KUKA KRL program: EPS_2_25252_SD4_A_20250910061725.src

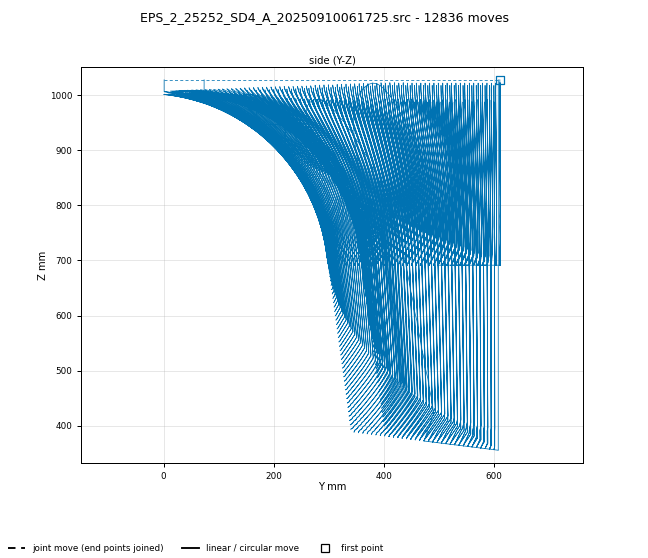
[picture p0: tool path of EPS_2_25252_SD4_A_20250910061725.src, 12836 of 12838 moves have a stored position in this frame; points joined in program order, loops and branches not executed]
&ACCESS RVP
&REL 4
&COMMENT QRS 19112012
&PARAM EDITMASK = *
DEF PART()
EXT BAS (BAS_COMMAND :IN,REAL :IN )
INT I
BAS (#INITMOV,0 )

;KUKA QRS Post kuka4.cps  Date:22-06-2017 !

File_ID=2825

QRS_PRE_INIT()

;Init var - Until changes are made in qrs_pre_init
Outlet_Square_prg=0
Inlet_1_Square_prg=0
Inlet_2_Square_prg=0
Inlet_3_Square_prg=0
Inlet_4_Square_prg=0
Inlet_5_Square_prg=0

Outlet_1={X 0.000, Y 400.000, Z 713.000, B 0.000, E1 0.000 }
Inlet_1={X 0.000, Y 400.000, Z 683.000, B 0.000, E1 208.000 }
Outlet_1_type=610
Inlet_1_type=610
;QRS#1=Sidecore dimensions
;QRS#2=600-24" Concrete
;QRS#3=600-24" Concrete
;QRS#4=
;QRS#5=
;QRS#6=
;QRS#7=
;QRS#8=
;QRS#9=S306-34L
;QRS#10=S306-34L
;QRS#11=
;QRS#12=
;QRS#13=
;QRS#14=
;QRS#15=
;QRS#16=1220x127x1372 4,5'
;QRS#17=EPS Height
;QRS#18=1018
;QRS#19=*
;QRS#20= UPDATED VERSION 22-06-2017
;QRS#21=*
Outlet_Square=0450
Inlet_1_Square=0450
Inlet_2_Square=0
Inlet_3_Square=0
Inlet_4_Square=0
Inlet_5_Square=0
Mill_Square=1
Outlet_Square_Prg=264
Inlet_1_Square_prg=264

QRS_INIT()

$ADVANCE=5

; T1
PTP {E1 178.274,E2 178.274}
PTP {X 0,Y 610.745,A -85,B 0,C 180,E1 178.274,E2 178.274,E3 0,E4 0,E5 0,E6 0}
QRS_SPEED_INIT()
LIN {X 0,Y 610.745,Z 1028,A -85,B 0,C 180,E1 178.274,E2 178.274,E3 0,E4 0,E5 0,E6 0} C_VEL
LIN {X 0,Y 610.745,Z 693.44,A -85,B 0,C 180,E1 178.274,E2 178.274} C_VEL
LIN {X 0,Y 610.771,Z 691.44,A -85,B 0,C 180,E1 178.462,E2 178.462} C_VEL
LIN {X 0,Y 611.874,Z 691.44,A -85,B 0,C 180,E1 181.167,E2 181.167} C_VEL
LIN {X 0,Y 611.801,Z 691.44,A -85,B 0,C 180,E1 188.197,E2 188.197} C_VEL
LIN {X 0,Y 611.817,Z 691.44,A -85,B 0,C 180,E1 195.354,E2 195.354} C_VEL
LIN {X 0,Y 611.765,Z 691.44,A -85,B 0,C 180,E1 202.769,E2 202.769} C_VEL
LIN {X 0,Y 611.741,Z 691.44,A -85,B 0,C 180,E1 210.614,E2 210.614} C_VEL
LIN {X 0,Y 610.574,Z 691.44,A -85,B 0,C 180,E1 217.262,E2 217.262} C_VEL
LIN {X 0,Y 611.71,Z 691.44,A -85,B 0,C 180,E1 219.162,E2 219.162} C_VEL
LIN {X 0,Y 610.308,Z 691.44,A -85,B 0,C 180,E1 222.361,E2 222.361} C_VEL
LIN {X 0,Y 610.623,Z 691.44,A -85,B 0,C 180,E1 225.583,E2 225.583} C_VEL
LIN {X 0,Y 611.712,Z 691.44,A -85,B 0,C 180,E1 227.765,E2 227.765} C_VEL
LIN {X 0,Y 611.694,Z 691.44,A -85,B 0,C 180,E1 235.934,E2 235.934} C_VEL
LIN {X 0,Y 611.734,Z 691.44,A -85,B 0,C 180,E1 236.288,E2 236.288} C_VEL
LIN {X 0,Y 610.695,Z 691.44,A -85,B 0,C 180,E1 236.459,E2 236.459} C_VEL
LIN {X 0,Y 610.433,Z 691.491,A -85,B 0,C 180,E1 236.481,E2 236.481} C_VEL
LIN {X 0,Y 611.42,Z 731.428,A -85,B 0,C 180,E1 237.097,E2 237.097} C_VEL
LIN {X 0,Y 611.517,Z 745.268,A -85,B 0,C 180,E1 237.335,E2 237.335} C_VEL
LIN {X 0,Y 611.325,Z 761.349,A -85,B 0,C 180,E1 237.681,E2 237.681} C_VEL
LIN {X 0,Y 611.672,Z 775.491,A -85,B 0,C 180,E1 238.087,E2 238.087} C_VEL
LIN {X 0,Y 611.736,Z 790.25,A -85,B 0,C 180,E1 238.571,E2 238.571} C_VEL
LIN {X 0,Y 611.693,Z 805.413,A -85,B 0,C 180,E1 239.145,E2 239.145} C_VEL
LIN {X 0,Y 611.448,Z 819.873,A -85,B 0,C 180,E1 239.763,E2 239.763} C_VEL
LIN {X 0,Y 611.625,Z 833.383,A -85,B 0,C 180,E1 240.435,E2 240.435} C_VEL
LIN {X 0,Y 611.599,Z 846.987,A -85,B 0,C 180,E1 241.179,E2 241.179} C_VEL
LIN {X 0,Y 611.634,Z 859.687,A -85,B 0,C 180,E1 241.947,E2 241.947} C_VEL
LIN {X 0,Y 611.641,Z 873.337,A -85,B 0,C 180,E1 242.859,E2 242.859} C_VEL
LIN {X 0,Y 611.572,Z 885.154,A -85,B 0,C 180,E1 243.716,E2 243.716} C_VEL
LIN {X 0,Y 611.333,Z 897.162,A -85,B 0,C 180,E1 244.66,E2 244.66} C_VEL
LIN {X 0,Y 611.276,Z 908.948,A -85,B 0,C 180,E1 245.678,E2 245.678} C_VEL
LIN {X 0,Y 611.472,Z 919.359,A -85,B 0,C 180,E1 246.662,E2 246.662} C_VEL
LIN {X 0,Y 611.734,Z 929.987,A -85,B 0,C 180,E1 247.753,E2 247.753} C_VEL
LIN {X 0,Y 611.445,Z 939.605,A -85,B 0,C 180,E1 248.799,E2 248.799} C_VEL
LIN {X 0,Y 611.088,Z 948.776,A -85,B 0,C 180,E1 249.876,E2 249.876} C_VEL
LIN {X 0,Y 611.074,Z 958.333,A -85,B 0,C 180,E1 251.115,E2 251.115} C_VEL
LIN {X 0,Y 611.399,Z 966.018,A -85,B 0,C 180,E1 252.202,E2 252.202} C_VEL
LIN {X 0,Y 611.821,Z 973.294,A -85,B 0,C 180,E1 253.324,E2 253.324} C_VEL
LIN {X 0,Y 611.107,Z 982.506,A -85,B 0,C 180,E1 254.862,E2 254.862} C_VEL
LIN {X 0,Y 610.739,Z 989.282,A -85,B 0,C 180,E1 256.13,E2 256.13} C_VEL
LIN {X 0,Y 610.875,Z 995.066,A -85,B 0,C 180,E1 257.336,E2 257.336} C_VEL
LIN {X 0,Y 611.566,Z 1001.375,A -85,B 0,C 180,E1 258.842,E2 258.842} C_VEL
LIN {X 0,Y 611.85,Z 1003.595,A -85,B 0,C 180,E1 259.441,E2 259.441} C_VEL
LIN {X 0,Y 611.525,Z 1005.814,A -85,B 0,C 180,E1 260.029,E2 260.029} C_VEL
LIN {X 0,Y 610.929,Z 1009.655,A -85,B 0,C 180,E1 261.204,E2 261.204} C_VEL
LIN {X 0,Y 610.672,Z 1012.99,A -85,B 0,C 180,E1 262.381,E2 262.381} C_VEL
LIN {X 0,Y 610.672,Z 1014.551,A -85,B 0,C 180,E1 262.97,E2 262.97} C_VEL
LIN {X 0,Y 611.06,Z 1017.123,A -85,B 0,C 180,E1 264.151,E2 264.151} C_VEL
LIN {X 0,Y 611.711,Z 1019.175,A -85,B 0,C 180,E1 265.329,E2 265.329} C_VEL
LIN {X 0,Y 611.37,Z 1020.807,A -85,B 0,C 180,E1 266.497,E2 266.497} C_VEL
LIN {X 0,Y 610.858,Z 1021.972,A -85,B 0,C 180,E1 267.634,E2 267.634} C_VEL
LIN {X 0,Y 610.688,Z 1022.778,A -85,B 0,C 180,E1 269.07,E2 269.07} C_VEL
LIN {X 0,Y 611.538,Z 1022.689,A -85,B 0,C 180,E1 271.17,E2 271.17} C_VEL
LIN {X 0,Y 611.319,Z 1021.671,A -85,B 0,C 180,E1 272.765,E2 272.765} C_VEL
LIN {X 0,Y 611.035,Z 1020.812,A -85,B 0,C 180,E1 273.51,E2 273.51} C_VEL
LIN {X 0,Y 610.805,Z 1019.194,A -85,B 0,C 180,E1 274.684,E2 274.684} C_VEL
LIN {X 0,Y 611.004,Z 1017.111,A -85,B 0,C 180,E1 275.855,E2 275.855} C_VEL
LIN {X 0,Y 611.55,Z 1014.527,A -85,B 0,C 180,E1 277.025,E2 277.025} C_VEL
LIN {X 0,Y 611.873,Z 1012.959,A -85,B 0,C 180,E1 277.61,E2 277.61} C_VEL
LIN {X 0,Y 611.24,Z 1009.637,A -85,B 0,C 180,E1 278.798,E2 278.798} C_VEL
LIN {X 0,Y 610.738,Z 1005.793,A -85,B 0,C 180,E1 279.99,E2 279.99} C_VEL
LIN {X 0,Y 610.738,Z 1000.147,A -85,B 0,C 180,E1 281.477,E2 281.477} C_VEL
LIN {X 0,Y 611.2,Z 995.039,A -85,B 0,C 180,E1 282.663,E2 282.663} C_VEL
LIN {X 0,Y 611.828,Z 989.347,A -85,B 0,C 180,E1 283.832,E2 283.832} C_VEL
LIN {X 0,Y 611.263,Z 982.264,A -85,B 0,C 180,E1 285.179,E2 285.179} C_VEL
LIN {X 0,Y 610.874,Z 973.74,A -85,B 0,C 180,E1 286.634,E2 286.634} C_VEL
LIN {X 0,Y 611.107,Z 964.915,A -85,B 0,C 180,E1 287.966,E2 287.966} C_VEL
LIN {X 0,Y 611.627,Z 956.003,A -85,B 0,C 180,E1 289.182,E2 289.182} C_VEL
LIN {X 0,Y 611.763,Z 951.154,A -85,B 0,C 180,E1 289.796,E2 289.796} C_VEL
LIN {X 0,Y 611.529,Z 944.981,A -85,B 0,C 180,E1 290.566,E2 290.566} C_VEL
LIN {X 0,Y 611.268,Z 937.362,A -85,B 0,C 180,E1 291.465,E2 291.465} C_VEL
LIN {X 0,Y 611.182,Z 926.922,A -85,B 0,C 180,E1 292.59,E2 292.59} C_VEL
LIN {X 0,Y 611.438,Z 916.306,A -85,B 0,C 180,E1 293.633,E2 293.633} C_VEL
LIN {X 0,Y 611.68,Z 905.113,A -85,B 0,C 180,E1 294.645,E2 294.645} C_VEL
LIN {X 0,Y 611.642,Z 894.625,A -85,B 0,C 180,E1 295.535,E2 295.535} C_VEL
LIN {X 0,Y 611.47,Z 882.903,A -85,B 0,C 180,E1 296.459,E2 296.459} C_VEL
LIN {X 0,Y 611.456,Z 869.526,A -85,B 0,C 180,E1 297.413,E2 297.413} C_VEL
LIN {X 0,Y 611.583,Z 857.642,A -85,B 0,C 180,E1 298.184,E2 298.184} C_VEL
LIN {X 0,Y 611.506,Z 843.831,A -85,B 0,C 180,E1 299.006,E2 299.006} C_VEL
LIN {X 0,Y 611.705,Z 829.665,A -85,B 0,C 180,E1 299.75,E2 299.75} C_VEL
LIN {X 0,Y 611.695,Z 816.017,A -85,B 0,C 180,E1 300.401,E2 300.401} C_VEL
LIN {X 0,Y 611.697,Z 800.985,A -85,B 0,C 180,E1 301.031,E2 301.031} C_VEL
LIN {X 0,Y 611.541,Z 786.836,A -85,B 0,C 180,E1 301.558,E2 301.558} C_VEL
LIN {X 0,Y 611.397,Z 780.445,A -85,B 0,C 180,E1 301.77,E2 301.77} C_VEL
LIN {X 0,Y 611.688,Z 770.796,A -85,B 0,C 180,E1 302.045,E2 302.045} C_VEL
LIN {X 0,Y 611.796,Z 757.518,A -85,B 0,C 180,E1 302.385,E2 302.385} C_VEL
LIN {X 0,Y 611.771,Z 741.883,A -85,B 0,C 180,E1 302.711,E2 302.711} C_VEL
LIN {X 0,Y 611.529,Z 722.323,A -85,B 0,C 180,E1 303.027,E2 303.027} C_VEL
LIN {X 0,Y 610.568,Z 694.458,A -85,B 0,C 180,E1 303.469,E2 303.469} C_VEL
LIN {X 0,Y 610.459,Z 691.44,A -85,B 0,C 180,E1 303.523,E2 303.523} C_VEL
LIN {X 0,Y 610.921,Z 691.44,A -85,B 0,C 180,E1 303.566,E2 303.566} C_VEL
LIN {X 0,Y 611.586,Z 691.44,A -85,B 0,C 180,E1 303.671,E2 303.671} C_VEL
LIN {X 0,Y 611.829,Z 691.44,A -85,B 0,C 180,E1 303.949,E2 303.949} C_VEL
LIN {X 0,Y 611.808,Z 691.44,A -85,B 0,C 180,E1 309.156,E2 309.156} C_VEL
LIN {X 0,Y 610.369,Z 691.44,A -85,B 0,C 180,E1 312.357,E2 312.357} C_VEL
LIN {X 0,Y 610.678,Z 691.44,A -85,B 0,C 180,E1 315.579,E2 315.579} C_VEL
LIN {X 0,Y 611.761,Z 691.44,A -85,B 0,C 180,E1 317.763,E2 317.763} C_VEL
LIN {X 0,Y 610.246,Z 691.44,A -85,B 0,C 180,E1 323.688,E2 323.688} C_VEL
LIN {X 0,Y 611.757,Z 691.44,A -85,B 0,C 180,E1 326.634,E2 326.634} C_VEL
LIN {X 0,Y 611.785,Z 691.44,A -85,B 0,C 180,E1 334.675,E2 334.675} C_VEL
LIN {X 0,Y 611.513,Z 691.44,A -85,B 0,C 180,E1 343.29,E2 343.29} C_VEL
LIN {X 0,Y 611.276,Z 691.44,A -85,B 0,C 180,E1 344.632,E2 344.632} C_VEL
LIN {X 0,Y 611.855,Z 691.44,A -85,B 0,C 180,E1 351.804,E2 351.804} C_VEL
LIN {X 0,Y 611.868,Z 691.44,A -85,B 0,C 180,E1 358.833,E2 358.833} C_VEL
LIN {X 0,Y 611.856,Z 691.44,A -85,B 0,C 180,E1 365.845,E2 365.845} C_VEL
LIN {X 0,Y 611.824,Z 691.44,A -85,B 0,C 180,E1 372.947,E2 372.947} C_VEL
LIN {X 0,Y 611.839,Z 691.44,A -85,B 0,C 180,E1 380.258,E2 380.258} C_VEL
LIN {X 0,Y 611.447,Z 691.44,A -85,B 0,C 180,E1 387.953,E2 387.953} C_VEL
LIN {X 0,Y 611.305,Z 691.44,A -85,B 0,C 180,E1 388.77,E2 388.77} C_VEL
LIN {X 0,Y 610.886,Z 691.44,A -85,B 0,C 180,E1 388.826,E2 388.826} C_VEL
LIN {X 0,Y 610.605,Z 692.257,A -85,B 0,C 180,E1 388.871,E2 388.871} C_VEL
LIN {X 0,Y 611.169,Z 709.751,A -85,B 0,C 180,E1 389.172,E2 389.172} C_VEL
LIN {X 0,Y 611.314,Z 717.452,A -85,B 0,C 180,E1 389.324,E2 389.324} C_VEL
LIN {X 0,Y 611.678,Z 731.173,A -85,B 0,C 180,E1 389.652,E2 389.652} C_VEL
LIN {X 0,Y 611.747,Z 746.429,A -85,B 0,C 180,E1 390.076,E2 390.076} C_VEL
LIN {X 0,Y 611.722,Z 761.243,A -85,B 0,C 180,E1 390.562,E2 390.562} C_VEL
LIN {X 0,Y 611.499,Z 775.09,A -85,B 0,C 180,E1 391.075,E2 391.075} C_VEL
LIN {X 0,Y 611.473,Z 779.918,A -85,B 0,C 180,E1 391.281,E2 391.281} C_VEL
LIN {X 0,Y 611.645,Z 790.127,A -85,B 0,C 180,E1 391.74,E2 391.74} C_VEL
LIN {X 0,Y 611.609,Z 803.759,A -85,B 0,C 180,E1 392.409,E2 392.409} C_VEL
LIN {X 0,Y 611.603,Z 816.719,A -85,B 0,C 180,E1 393.117,E2 393.117} C_VEL
LIN {X 0,Y 611.675,Z 830.91,A -85,B 0,C 180,E1 393.985,E2 393.985} C_VEL
LIN {X 0,Y 611.602,Z 842.971,A -85,B 0,C 180,E1 394.785,E2 394.785} C_VEL
LIN {X 0,Y 611.498,Z 854.83,A -85,B 0,C 180,E1 395.642,E2 395.642} C_VEL
LIN {X 0,Y 611.307,Z 867.776,A -85,B 0,C 180,E1 396.666,E2 396.666} C_VEL
LIN {X 0,Y 611.372,Z 878.558,A -85,B 0,C 180,E1 397.601,E2 397.601} C_VEL
LIN {X 0,Y 611.624,Z 890.243,A -85,B 0,C 180,E1 398.712,E2 398.712} C_VEL
LIN {X 0,Y 611.707,Z 898.191,A -85,B 0,C 180,E1 399.512,E2 399.512} C_VEL
LIN {X 0,Y 611.316,Z 909.19,A -85,B 0,C 180,E1 400.7,E2 400.7} C_VEL
LIN {X 0,Y 611.099,Z 918.7,A -85,B 0,C 180,E1 401.821,E2 401.821} C_VEL
LIN {X 0,Y 611.248,Z 927.831,A -85,B 0,C 180,E1 403.005,E2 403.005} C_VEL
LIN {X 0,Y 611.668,Z 936.135,A -85,B 0,C 180,E1 404.183,E2 404.183} C_VEL
LIN {X 0,Y 611.824,Z 939.64,A -85,B 0,C 180,E1 404.723,E2 404.723} C_VEL
LIN {X 0,Y 611.451,Z 944.743,A -85,B 0,C 180,E1 405.504,E2 405.504} C_VEL
LIN {X 0,Y 610.879,Z 952.592,A -85,B 0,C 180,E1 406.827,E2 406.827} C_VEL
LIN {X 0,Y 610.763,Z 958.932,A -85,B 0,C 180,E1 408.012,E2 408.012} C_VEL
LIN {X 0,Y 611.164,Z 965.191,A -85,B 0,C 180,E1 409.325,E2 409.325} C_VEL
LIN {X 0,Y 611.749,Z 970.163,A -85,B 0,C 180,E1 410.501,E2 410.501} C_VEL
LIN {X 0,Y 611.799,Z 971.533,A -85,B 0,C 180,E1 410.843,E2 410.843} C_VEL
LIN {X 0,Y 611.094,Z 976.54,A -85,B 0,C 180,E1 412.191,E2 412.191} C_VEL
LIN {X 0,Y 610.689,Z 981.321,A -85,B 0,C 180,E1 413.717,E2 413.717} C_VEL
LIN {X 0,Y 610.828,Z 984.007,A -85,B 0,C 180,E1 414.715,E2 414.715} C_VEL
LIN {X 0,Y 611.36,Z 986.671,A -85,B 0,C 180,E1 415.906,E2 415.906} C_VEL
LIN {X 0,Y 611.759,Z 988.072,A -85,B 0,C 180,E1 416.632,E2 416.632} C_VEL
LIN {X 0,Y 611.578,Z 989.364,A -85,B 0,C 180,E1 417.391,E2 417.391} C_VEL
LIN {X 0,Y 611.173,Z 990.338,A -85,B 0,C 180,E1 418.053,E2 418.053} C_VEL
LIN {X 0,Y 610.615,Z 991.788,A -85,B 0,C 180,E1 419.321,E2 419.321} C_VEL
LIN {X 0,Y 610.523,Z 992.469,A -85,B 0,C 180,E1 420.272,E2 420.272} C_VEL
LIN {X 0,Y 611.094,Z 992.97,A -85,B 0,C 180,E1 422.028,E2 422.028} C_VEL
LIN {X 0,Y 611.703,Z 992.701,A -85,B 0,C 180,E1 423.035,E2 423.035} C_VEL
LIN {X 0,Y 611.246,Z 991.725,A -85,B 0,C 180,E1 424.65,E2 424.65} C_VEL
LIN {X 0,Y 611.014,Z 990.672,A -85,B 0,C 180,E1 425.583,E2 425.583} C_VEL
LIN {X 0,Y 611.041,Z 989.261,A -85,B 0,C 180,E1 426.594,E2 426.594} C_VEL
LIN {X 0,Y 611.469,Z 986.875,A -85,B 0,C 180,E1 427.909,E2 427.909} C_VEL
LIN {X 0,Y 611.718,Z 985.672,A -85,B 0,C 180,E1 428.452,E2 428.452} C_VEL
LIN {X 0,Y 611.671,Z 984.243,A -85,B 0,C 180,E1 429.094,E2 429.094} C_VEL
LIN {X 0,Y 611.022,Z 980.931,A -85,B 0,C 180,E1 430.334,E2 430.334} C_VEL
LIN {X 0,Y 610.678,Z 976.08,A -85,B 0,C 180,E1 431.867,E2 431.867} C_VEL
LIN {X 0,Y 611.102,Z 970.181,A -85,B 0,C 180,E1 433.417,E2 433.417} C_VEL
LIN {X 0,Y 611.736,Z 964.877,A -85,B 0,C 180,E1 434.642,E2 434.642} C_VEL
LIN {X 0,Y 611.869,Z 963.707,A -85,B 0,C 180,E1 434.881,E2 434.881} C_VEL
LIN {X 0,Y 611.295,Z 957.857,A -85,B 0,C 180,E1 436.093,E2 436.093} C_VEL
LIN {X 0,Y 610.844,Z 951.248,A -85,B 0,C 180,E1 437.33,E2 437.33} C_VEL
LIN {X 0,Y 610.861,Z 944.132,A -85,B 0,C 180,E1 438.525,E2 438.525} C_VEL
LIN {X 0,Y 611.442,Z 934.12,A -85,B 0,C 180,E1 440.022,E2 440.022} C_VEL
LIN {X 0,Y 611.779,Z 927.636,A -85,B 0,C 180,E1 440.915,E2 440.915} C_VEL
LIN {X 0,Y 611.298,Z 916.221,A -85,B 0,C 180,E1 442.383,E2 442.383} C_VEL
LIN {X 0,Y 611.105,Z 907.499,A -85,B 0,C 180,E1 443.411,E2 443.411} C_VEL
LIN {X 0,Y 611.276,Z 896.469,A -85,B 0,C 180,E1 444.587,E2 444.587} C_VEL
LIN {X 0,Y 611.607,Z 885.785,A -85,B 0,C 180,E1 445.629,E2 445.629} C_VEL
LIN {X 0,Y 611.677,Z 874.98,A -85,B 0,C 180,E1 446.612,E2 446.612} C_VEL
LIN {X 0,Y 611.482,Z 863.577,A -85,B 0,C 180,E1 447.58,E2 447.58} C_VEL
LIN {X 0,Y 611.387,Z 852.606,A -85,B 0,C 180,E1 448.44,E2 448.44} C_VEL
LIN {X 0,Y 611.511,Z 840.572,A -85,B 0,C 180,E1 449.297,E2 449.297} C_VEL
LIN {X 0,Y 611.618,Z 828.032,A -85,B 0,C 180,E1 450.114,E2 450.114} C_VEL
LIN {X 0,Y 611.589,Z 820.26,A -85,B 0,C 180,E1 450.581,E2 450.581} C_VEL
LIN {X 0,Y 611.69,Z 812.057,A -85,B 0,C 180,E1 451.048,E2 451.048} C_VEL
LIN {X 0,Y 611.688,Z 799.787,A -85,B 0,C 180,E1 451.7,E2 451.7} C_VEL
LIN {X 0,Y 611.688,Z 786.561,A -85,B 0,C 180,E1 452.333,E2 452.333} C_VEL
LIN {X 0,Y 611.606,Z 770.8,A -85,B 0,C 180,E1 452.998,E2 452.998} C_VEL
LIN {X 0,Y 611.452,Z 760.468,A -85,B 0,C 180,E1 453.393,E2 453.393} C_VEL
LIN {X 0,Y 611.779,Z 742.741,A -85,B 0,C 180,E1 453.944,E2 453.944} C_VEL
LIN {X 0,Y 611.784,Z 726.733,A -85,B 0,C 180,E1 454.359,E2 454.359} C_VEL
LIN {X 0,Y 611.687,Z 711.157,A -85,B 0,C 180,E1 454.684,E2 454.684} C_VEL
LIN {X 0,Y 611.139,Z 694.076,A -85,B 0,C 180,E1 454.981,E2 454.981} C_VEL
LIN {X 0,Y 611.034,Z 691.44,A -85,B 0,C 180,E1 455.033,E2 455.033} C_VEL
LIN {X 0,Y 611.614,Z 691.44,A -85,B 0,C 180,E1 455.13,E2 455.13} C_VEL
LIN {X 0,Y 611.882,Z 691.44,A -85,B 0,C 180,E1 455.281,E2 455.281} C_VEL
LIN {X 0,Y 611.878,Z 691.44,A -85,B 0,C 180,E1 458.193,E2 458.193} C_VEL
LIN {X 0,Y 611.842,Z 691.44,A -85,B 0,C 180,E1 465.35,E2 465.35} C_VEL
LIN {X 0,Y 611.83,Z 691.44,A -85,B 0,C 180,E1 472.763,E2 472.763} C_VEL
LIN {X 0,Y 611.802,Z 691.44,A -85,B 0,C 180,E1 480.606,E2 480.606} C_VEL
LIN {X 0,Y 610.636,Z 691.44,A -85,B 0,C 180,E1 487.261,E2 487.261} C_VEL
LIN {X 0,Y 611.766,Z 691.44,A -85,B 0,C 180,E1 489.152,E2 489.152} C_VEL
LIN {X 0,Y 610.361,Z 691.44,A -85,B 0,C 180,E1 492.35,E2 492.35} C_VEL
LIN {X 0,Y 610.672,Z 691.44,A -85,B 0,C 180,E1 495.572,E2 495.572} C_VEL
LIN {X 0,Y 611.767,Z 691.44,A -85,B 0,C 180,E1 497.763,E2 497.763} C_VEL
LIN {X 0,Y 610.277,Z 691.44,A -85,B 0,C 180,E1 503.69,E2 503.69} C_VEL
LIN {X 0,Y 611.793,Z 691.44,A -85,B 0,C 180,E1 506.636,E2 506.636} C_VEL
LIN {X 0,Y 611.817,Z 691.44,A -85,B 0,C 180,E1 514.677,E2 514.677} C_VEL
LIN {X 0,Y 611.476,Z 691.44,A -85,B 0,C 180,E1 523.282,E2 523.282} C_VEL
LIN {X 0,Y 611.637,Z 691.44,A -85,B 0,C 180,E1 524.641,E2 524.641} C_VEL
LIN {X 0,Y 611.854,Z 691.44,A -85,B 0,C 180,E1 527.054,E2 527.054} C_VEL
LIN {X 0,Y 611.811,Z 691.44,A -85,B 0,C 180,E1 534.155,E2 534.155} C_VEL
LIN {X 0,Y 610.771,Z 691.44,A -85,B 0,C 180,E1 538.462,E2 538.462} C_VEL
LIN {X 0,Y 603.352,Z 691.44,A -85,B 0,C 180,E1 541.754,E2 541.754} C_VEL
LIN {X 0,Y 603.133,Z 691.44,A -85,B 0,C 180,E1 549.4,E2 549.4} C_VEL
LIN {X 0,Y 603.021,Z 691.44,A -85,B 0,C 180,E1 556.806,E2 556.806} C_VEL
LIN {X 0,Y 602.764,Z 691.44,A -85,B 0,C 180,E1 564.526,E2 564.526} C_VEL
LIN {X 0,Y 602.607,Z 691.44,A -85,B 0,C 180,E1 572.471,E2 572.471} C_VEL
LIN {X 0,Y 603.228,Z 691.44,A -85,B 0,C 180,E1 579.886,E2 579.886} C_VEL
LIN {X 0,Y 603.381,Z 691.44,A -85,B 0,C 180,E1 588.201,E2 588.201} C_VEL
LIN {X 0,Y 603.771,Z 692.599,A -85,B 0,C 180,E1 596.077,E2 596.077} C_VEL
LIN {X 0,Y 604.811,Z 776.815,A -85,B 0,C 180,E1 597.724,E2 597.724} C_VEL
LIN {X 0,Y 604.426,Z 842.241,A -85,B 0,C 180,E1 600.534,E2 600.534} C_VEL
LIN {X 0,Y 603.773,Z 901.578,A -85,B 0,C 180,E1 604.704,E2 604.704} C_VEL
LIN {X 0,Y 603.28,Z 950.003,A -85,B 0,C 180,E1 609.764,E2 609.764} C_VEL
LIN {X 0,Y 603.004,Z 985.712,A -85,B 0,C 180,E1 615.259,E2 615.259} C_VEL
LIN {X 0,Y 603.039,Z 1009.22,A -85,B 0,C 180,E1 620.95,E2 620.95} C_VEL
LIN {X 0,Y 603.404,Z 1020.765,A -85,B 0,C 180,E1 626.395,E2 626.395} C_VEL
LIN {X 0,Y 603.378,Z 1022.148,A -85,B 0,C 180,E1 632.162,E2 632.162} C_VEL
LIN {X 0,Y 603.3,Z 1010.379,A -85,B 0,C 180,E1 638.68,E2 638.68} C_VEL
LIN {X 0,Y 603.371,Z 983.789,A -85,B 0,C 180,E1 645.095,E2 645.095} C_VEL
LIN {X 0,Y 603.641,Z 943.759,A -85,B 0,C 180,E1 650.993,E2 650.993} C_VEL
LIN {X 0,Y 604.095,Z 892.092,A -85,B 0,C 180,E1 656.08,E2 656.08} C_VEL
LIN {X 0,Y 604.594,Z 831.211,A -85,B 0,C 180,E1 660.06,E2 660.06} C_VEL
LIN {X 0,Y 604.93,Z 766.154,A -85,B 0,C 180,E1 662.573,E2 662.573} C_VEL
LIN {X 0,Y 603.81,Z 691.44,A -85,B 0,C 180,E1 663.958,E2 663.958} C_VEL
LIN {X 0,Y 602.445,Z 691.44,A -85,B 0,C 180,E1 672.039,E2 672.039} C_VEL
LIN {X 0,Y 603.392,Z 691.44,A -85,B 0,C 180,E1 678.234,E2 678.234} C_VEL
LIN {X 0,Y 603.213,Z 691.44,A -85,B 0,C 180,E1 687.437,E2 687.437} C_VEL
LIN {X 0,Y 603.151,Z 691.44,A -85,B 0,C 180,E1 695.491,E2 695.491} C_VEL
LIN {X 0,Y 603.231,Z 691.44,A -85,B 0,C 180,E1 704.699,E2 704.699} C_VEL
LIN {X 0,Y 602.905,Z 691.44,A -85,B 0,C 180,E1 713.859,E2 713.859} C_VEL
LIN {X 0,Y 602.969,Z 691.44,A -85,B 0,C 180,E1 720.731,E2 720.731} C_VEL
LIN {X 0,Y 602.865,Z 691.44,A -85,B 0,C 180,E1 727.965,E2 727.965} C_VEL
LIN {X 0,Y 602.759,Z 691.44,A -85,B 0,C 180,E1 735.334,E2 735.334} C_VEL
LIN {X 0,Y 603.099,Z 691.44,A -85,B 0,C 180,E1 741.402,E2 741.402} C_VEL
LIN {X 0,Y 603.488,Z 692.92,A -85,B 0,C 180,E1 748.439,E2 748.439} C_VEL
LIN {X 0,Y 604.771,Z 763.762,A -85,B 0,C 180,E1 750.254,E2 750.254} C_VEL
LIN {X 0,Y 604.392,Z 826.547,A -85,B 0,C 180,E1 753.338,E2 753.338} C_VEL
LIN {X 0,Y 603.829,Z 884.4,A -85,B 0,C 180,E1 757.827,E2 757.827} C_VEL
LIN {X 0,Y 603.494,Z 931.716,A -85,B 0,C 180,E1 763.302,E2 763.302} C_VEL
LIN {X 0,Y 603.25,Z 966.27,A -85,B 0,C 180,E1 769.413,E2 769.413} C_VEL
LIN {X 0,Y 603.181,Z 986.033,A -85,B 0,C 180,E1 775.522,E2 775.522} C_VEL
LIN {X 0,Y 602.596,Z 992.687,A -85,B 0,C 180,E1 780.588,E2 780.588} C_VEL
LIN {X 0,Y 603.035,Z 990.881,A -85,B 0,C 180,E1 785.466,E2 785.466} C_VEL
LIN {X 0,Y 602.914,Z 980.226,A -85,B 0,C 180,E1 790.69,E2 790.69} C_VEL
LIN {X 0,Y 603.177,Z 956.506,A -85,B 0,C 180,E1 796.542,E2 796.542} C_VEL
LIN {X 0,Y 603.526,Z 918.219,A -85,B 0,C 180,E1 802.415,E2 802.415} C_VEL
LIN {X 0,Y 604.007,Z 865.701,A -85,B 0,C 180,E1 807.75,E2 807.75} C_VEL
LIN {X 0,Y 604.561,Z 805.25,A -85,B 0,C 180,E1 811.798,E2 811.798} C_VEL
LIN {X 0,Y 604.945,Z 742.287,A -85,B 0,C 180,E1 814.361,E2 814.361} C_VEL
LIN {X 0,Y 603.831,Z 691.44,A -85,B 0,C 180,E1 815.589,E2 815.589} C_VEL
LIN {X 0,Y 603.817,Z 691.44,A -85,B 0,C 180,E1 825.302,E2 825.302} C_VEL
LIN {X 0,Y 602.819,Z 691.44,A -85,B 0,C 180,E1 834.544,E2 834.544} C_VEL
LIN {X 0,Y 602.655,Z 691.44,A -85,B 0,C 180,E1 842.493,E2 842.493} C_VEL
LIN {X 0,Y 603.28,Z 691.44,A -85,B 0,C 180,E1 849.902,E2 849.902} C_VEL
LIN {X 0,Y 603.413,Z 691.44,A -85,B 0,C 180,E1 858.209,E2 858.209} C_VEL
LIN {X 0,Y 603.274,Z 691.44,A -85,B 0,C 180,E1 867.429,E2 867.429} C_VEL
LIN {X 0,Y 603.222,Z 691.44,A -85,B 0,C 180,E1 875.472,E2 875.472} C_VEL
LIN {X 0,Y 603.68,Z 691.44,A -85,B 0,C 180,E1 886.178,E2 886.178} C_VEL
LIN {X 0,Y 603.355,Z 691.44,A -85,B 0,C 180,E1 894.941,E2 894.941} C_VEL
LIN {X 0,Y 603.352,Z 691.44,A -85,B 0,C 180,E1 901.754,E2 901.754} C_VEL
LIN {X 0,Y 594.726,Z 691.44,A -85,B 0,C 180,E1 905.048,E2 905.048} C_VEL
LIN {X 0,Y 594.678,Z 691.44,A -85,B 0,C 180,E1 911.02,E2 911.02} C_VEL
LIN {X 0,Y 594.935,Z 691.44,A -85,B 0,C 180,E1 917.042,E2 917.042} C_VEL
LIN {X 0,Y 594.592,Z 691.44,A -85,B 0,C 180,E1 925.031,E2 925.031} C_VEL
LIN {X 0,Y 595.114,Z 691.44,A -85,B 0,C 180,E1 931.494,E2 931.494} C_VEL
LIN {X 0,Y 594.616,Z 691.44,A -85,B 0,C 180,E1 941.157,E2 941.157} C_VEL
LIN {X 0,Y 594.701,Z 691.44,A -85,B 0,C 180,E1 949.403,E2 949.403} C_VEL
LIN {X 0,Y 595.542,Z 692.888,A -85,B 0,C 180,E1 955.547,E2 955.547} C_VEL
LIN {X 0,Y 597.96,Z 779.246,A -85,B 0,C 180,E1 957.389,E2 957.389} C_VEL
LIN {X 0,Y 597.256,Z 843.942,A -85,B 0,C 180,E1 960.239,E2 960.239} C_VEL
LIN {X 0,Y 596.217,Z 903.96,A -85,B 0,C 180,E1 964.57,E2 964.57} C_VEL
LIN {X 0,Y 595.472,Z 951.481,A -85,B 0,C 180,E1 969.681,E2 969.681} C_VEL
LIN {X 0,Y 595.078,Z 986.267,A -85,B 0,C 180,E1 975.164,E2 975.164} C_VEL
LIN {X 0,Y 594.98,Z 1010.376,A -85,B 0,C 180,E1 981.197,E2 981.197} C_VEL
LIN {X 0,Y 595.416,Z 1020.765,A -85,B 0,C 180,E1 986.346,E2 986.346} C_VEL
LIN {X 0,Y 595.363,Z 1022.149,A -85,B 0,C 180,E1 992.191,E2 992.191} C_VEL
LIN {X 0,Y 595.255,Z 1010.378,A -85,B 0,C 180,E1 998.799,E2 998.799} C_VEL
LIN {X 0,Y 595.436,Z 984.428,A -85,B 0,C 180,E1 1005.178,E2 1005.178} C_VEL
LIN {X 0,Y 595.87,Z 945.376,A -85,B 0,C 180,E1 1011.084,E2 1011.084} C_VEL
LIN {X 0,Y 596.621,Z 893.819,A -85,B 0,C 180,E1 1016.292,E2 1016.292} C_VEL
LIN {X 0,Y 597.479,Z 832.394,A -85,B 0,C 180,E1 1020.391,E2 1020.391} C_VEL
LIN {X 0,Y 598.13,Z 767.802,A -85,B 0,C 180,E1 1022.944,E2 1022.944} C_VEL
LIN {X 0,Y 595.595,Z 691.44,A -85,B 0,C 180,E1 1024.496,E2 1024.496} C_VEL
LIN {X 0,Y 594.336,Z 691.44,A -85,B 0,C 180,E1 1032.582,E2 1032.582} C_VEL
LIN {X 0,Y 594.664,Z 691.44,A -85,B 0,C 180,E1 1039.431,E2 1039.431} C_VEL
LIN {X 0,Y 594.713,Z 691.44,A -85,B 0,C 180,E1 1048.483,E2 1048.483} C_VEL
LIN {X 0,Y 594.493,Z 691.44,A -85,B 0,C 180,E1 1056.712,E2 1056.712} C_VEL
LIN {X 0,Y 595.239,Z 691.44,A -85,B 0,C 180,E1 1064.488,E2 1064.488} C_VEL
LIN {X 0,Y 595.057,Z 691.44,A -85,B 0,C 180,E1 1073.422,E2 1073.422} C_VEL
LIN {X 0,Y 594.978,Z 691.44,A -85,B 0,C 180,E1 1080.74,E2 1080.74} C_VEL
LIN {X 0,Y 594.836,Z 691.44,A -85,B 0,C 180,E1 1088.074,E2 1088.074} C_VEL
LIN {X 0,Y 594.71,Z 691.44,A -85,B 0,C 180,E1 1095.546,E2 1095.546} C_VEL
LIN {X 0,Y 594.927,Z 691.44,A -85,B 0,C 180,E1 1101.711,E2 1101.711} C_VEL
LIN {X 0,Y 595.452,Z 692.462,A -85,B 0,C 180,E1 1107.919,E2 1107.919} C_VEL
LIN {X 0,Y 597.927,Z 761.951,A -85,B 0,C 180,E1 1109.778,E2 1109.778} C_VEL
LIN {X 0,Y 597.153,Z 825.254,A -85,B 0,C 180,E1 1112.878,E2 1112.878} C_VEL
LIN {X 0,Y 596.153,Z 881.742,A -85,B 0,C 180,E1 1117.242,E2 1117.242} C_VEL
LIN {X 0,Y 595.526,Z 928.799,A -85,B 0,C 180,E1 1122.623,E2 1122.623} C_VEL
LIN {X 0,Y 594.978,Z 962.977,A -85,B 0,C 180,E1 1128.498,E2 1128.498} C_VEL
LIN {X 0,Y 594.762,Z 982.401,A -85,B 0,C 180,E1 1133.904,E2 1133.904} C_VEL
LIN {X 0,Y 594.841,Z 991.25,A -85,B 0,C 180,E1 1138.709,E2 1138.709} C_VEL
LIN {X 0,Y 595.078,Z 991.348,A -85,B 0,C 180,E1 1145.116,E2 1145.116} C_VEL
LIN {X 0,Y 594.873,Z 979.906,A -85,B 0,C 180,E1 1150.912,E2 1150.912} C_VEL
LIN {X 0,Y 595.199,Z 956.552,A -85,B 0,C 180,E1 1156.734,E2 1156.734} C_VEL
LIN {X 0,Y 595.713,Z 918.317,A -85,B 0,C 180,E1 1162.682,E2 1162.682} C_VEL
LIN {X 0,Y 596.503,Z 865.85,A -85,B 0,C 180,E1 1168.087,E2 1168.087} C_VEL
LIN {X 0,Y 597.429,Z 805.396,A -85,B 0,C 180,E1 1172.184,E2 1172.184} C_VEL
LIN {X 0,Y 598.172,Z 742.236,A -85,B 0,C 180,E1 1174.776,E2 1174.776} C_VEL
LIN {X 0,Y 595.767,Z 691.646,A -85,B 0,C 180,E1 1175.982,E2 1175.982} C_VEL
LIN {X 0,Y 595.668,Z 691.44,A -85,B 0,C 180,E1 1185.516,E2 1185.516} C_VEL
LIN {X 0,Y 594.686,Z 691.44,A -85,B 0,C 180,E1 1194.902,E2 1194.902} C_VEL
LIN {X 0,Y 595.159,Z 691.44,A -85,B 0,C 180,E1 1201.516,E2 1201.516} C_VEL
LIN {X 0,Y 594.674,Z 691.44,A -85,B 0,C 180,E1 1211.172,E2 1211.172} C_VEL
LIN {X 0,Y 594.684,Z 691.44,A -85,B 0,C 180,E1 1219.407,E2 1219.407} C_VEL
LIN {X 0,Y 594.782,Z 691.44,A -85,B 0,C 180,E1 1228.463,E2 1228.463} C_VEL
LIN {X 0,Y 594.503,Z 691.44,A -85,B 0,C 180,E1 1236.69,E2 1236.69} C_VEL
LIN {X 0,Y 595.653,Z 691.44,A -85,B 0,C 180,E1 1245.988,E2 1245.988} C_VEL
LIN {X 0,Y 595.369,Z 691.44,A -85,B 0,C 180,E1 1254.873,E2 1254.873} C_VEL
LIN {X 0,Y 595.304,Z 691.44,A -85,B 0,C 180,E1 1262.181,E2 1262.181} C_VEL
LIN {X 0,Y 594.726,Z 691.44,A -85,B 0,C 180,E1 1265.048,E2 1265.048} C_VEL
LIN {X 0,Y 587.444,Z 691.44,A -85,B 0,C 180,E1 1268.415,E2 1268.415} C_VEL
LIN {X 0,Y 586.846,Z 691.44,A -85,B 0,C 180,E1 1277.284,E2 1277.284} C_VEL
LIN {X 0,Y 586.536,Z 691.44,A -85,B 0,C 180,E1 1285.251,E2 1285.251} C_VEL
LIN {X 0,Y 586.482,Z 691.44,A -85,B 0,C 180,E1 1292.756,E2 1292.756} C_VEL
LIN {X 0,Y 586.581,Z 691.44,A -85,B 0,C 180,E1 1301.248,E2 1301.248} C_VEL
LIN {X 0,Y 587.044,Z 691.44,A -85,B 0,C 180,E1 1308.76,E2 1308.76} C_VEL
LIN {X 0,Y 587.273,Z 693.317,A -85,B 0,C 180,E1 1314.998,E2 1314.998} C_VEL
LIN {X 0,Y 590.809,Z 705.891,A -85,B 0,C 180,E1 1315.42,E2 1315.42} C_VEL
LIN {X 0,Y 591.136,Z 781.262,A -85,B 0,C 180,E1 1317.032,E2 1317.032} C_VEL
LIN {X 0,Y 590.118,Z 844.997,A -85,B 0,C 180,E1 1319.902,E2 1319.902} C_VEL
LIN {X 0,Y 588.714,Z 903.961,A -85,B 0,C 180,E1 1324.222,E2 1324.222} C_VEL
LIN {X 0,Y 587.671,Z 952.959,A -85,B 0,C 180,E1 1329.597,E2 1329.597} C_VEL
LIN {X 0,Y 587.106,Z 987.674,A -85,B 0,C 180,E1 1335.231,E2 1335.231} C_VEL
LIN {X 0,Y 587.027,Z 1010.376,A -85,B 0,C 180,E1 1341.076,E2 1341.076} C_VEL
LIN {X 0,Y 587.425,Z 1020.766,A -85,B 0,C 180,E1 1346.297,E2 1346.297} C_VEL
LIN {X 0,Y 587.349,Z 1022.149,A -85,B 0,C 180,E1 1352.221,E2 1352.221} C_VEL
LIN {X 0,Y 587.22,Z 1010.378,A -85,B 0,C 180,E1 1358.92,E2 1358.92} C_VEL
LIN {X 0,Y 587.436,Z 984.431,A -85,B 0,C 180,E1 1365.39,E2 1365.39} C_VEL
LIN {X 0,Y 588.113,Z 946.08,A -85,B 0,C 180,E1 1371.289,E2 1371.289} C_VEL
LIN {X 0,Y 589.148,Z 894.983,A -85,B 0,C 180,E1 1376.556,E2 1376.556} C_VEL
LIN {X 0,Y 590.365,Z 833.851,A -85,B 0,C 180,E1 1380.715,E2 1380.715} C_VEL
LIN {X 0,Y 591.343,Z 769.887,A -85,B 0,C 180,E1 1383.313,E2 1383.313} C_VEL
LIN {X 0,Y 589.008,Z 696.086,A -85,B 0,C 180,E1 1384.844,E2 1384.844} C_VEL
LIN {X 0,Y 587.411,Z 691.44,A -85,B 0,C 180,E1 1385.154,E2 1385.154} C_VEL
LIN {X 0,Y 586.299,Z 691.44,A -85,B 0,C 180,E1 1393.309,E2 1393.309} C_VEL
LIN {X 0,Y 586.544,Z 691.44,A -85,B 0,C 180,E1 1399.752,E2 1399.752} C_VEL
LIN {X 0,Y 586.784,Z 691.44,A -85,B 0,C 180,E1 1408.007,E2 1408.007} C_VEL
LIN {X 0,Y 586.505,Z 691.44,A -85,B 0,C 180,E1 1416.717,E2 1416.717} C_VEL
LIN {X 0,Y 587.22,Z 691.44,A -85,B 0,C 180,E1 1424.271,E2 1424.271} C_VEL
LIN {X 0,Y 587.08,Z 691.44,A -85,B 0,C 180,E1 1433.333,E2 1433.333} C_VEL
LIN {X 0,Y 586.973,Z 691.44,A -85,B 0,C 180,E1 1440.751,E2 1440.751} C_VEL
LIN {X 0,Y 586.828,Z 691.44,A -85,B 0,C 180,E1 1448.184,E2 1448.184} C_VEL
LIN {X 0,Y 586.674,Z 691.44,A -85,B 0,C 180,E1 1455.765,E2 1455.765} C_VEL
LIN {X 0,Y 586.776,Z 691.44,A -85,B 0,C 180,E1 1462.028,E2 1462.028} C_VEL
LIN {X 0,Y 587.221,Z 692.727,A -85,B 0,C 180,E1 1467.378,E2 1467.378} C_VEL
LIN {X 0,Y 591.008,Z 708.683,A -85,B 0,C 180,E1 1467.885,E2 1467.885} C_VEL
LIN {X 0,Y 590.652,Z 776.585,A -85,B 0,C 180,E1 1469.924,E2 1469.924} C_VEL
LIN {X 0,Y 589.663,Z 840.532,A -85,B 0,C 180,E1 1473.508,E2 1473.508} C_VEL
LIN {X 0,Y 588.641,Z 895.645,A -85,B 0,C 180,E1 1478.314,E2 1478.314} C_VEL
LIN {X 0,Y 588.07,Z 940.626,A -85,B 0,C 180,E1 1484.158,E2 1484.158} C_VEL
LIN {X 0,Y 587.731,Z 971.385,A -85,B 0,C 180,E1 1490.34,E2 1490.34} C_VEL
LIN {X 0,Y 587.519,Z 989.187,A -85,B 0,C 180,E1 1497.073,E2 1497.073} C_VEL
LIN {X 0,Y 587.356,Z 992.744,A -85,B 0,C 180,E1 1503.118,E2 1503.118} C_VEL
LIN {X 0,Y 587.369,Z 983.756,A -85,B 0,C 180,E1 1509.586,E2 1509.586} C_VEL
LIN {X 0,Y 587.467,Z 960.261,A -85,B 0,C 180,E1 1516.176,E2 1516.176} C_VEL
LIN {X 0,Y 587.981,Z 922.578,A -85,B 0,C 180,E1 1522.399,E2 1522.399} C_VEL
LIN {X 0,Y 588.962,Z 873.251,A -85,B 0,C 180,E1 1527.785,E2 1527.785} C_VEL
LIN {X 0,Y 590.212,Z 813.78,A -85,B 0,C 180,E1 1532.119,E2 1532.119} C_VEL
LIN {X 0,Y 591.211,Z 749.734,A -85,B 0,C 180,E1 1534.97,E2 1534.97} C_VEL
LIN {X 0,Y 589.42,Z 696.366,A -85,B 0,C 180,E1 1536.332,E2 1536.332} C_VEL
LIN {X 0,Y 587.703,Z 691.44,A -85,B 0,C 180,E1 1536.673,E2 1536.673} C_VEL
LIN {X 0,Y 587.54,Z 691.44,A -85,B 0,C 180,E1 1545.737,E2 1545.737} C_VEL
LIN {X 0,Y 587.26,Z 691.44,A -85,B 0,C 180,E1 1553.613,E2 1553.613} C_VEL
LIN {X 0,Y 586.861,Z 691.44,A -85,B 0,C 180,E1 1562.014,E2 1562.014} C_VEL
LIN {X 0,Y 586.637,Z 691.44,A -85,B 0,C 180,E1 1571.275,E2 1571.275} C_VEL
LIN {X 0,Y 587.059,Z 691.44,A -85,B 0,C 180,E1 1578.766,E2 1578.766} C_VEL
LIN {X 0,Y 586.844,Z 691.44,A -85,B 0,C 180,E1 1587.986,E2 1587.986} C_VEL
LIN {X 0,Y 586.481,Z 691.44,A -85,B 0,C 180,E1 1596.724,E2 1596.724} C_VEL
LIN {X 0,Y 587.623,Z 691.44,A -85,B 0,C 180,E1 1605.792,E2 1605.792} C_VEL
LIN {X 0,Y 587.362,Z 691.44,A -85,B 0,C 180,E1 1614.803,E2 1614.803} C_VEL
LIN {X 0,Y 587.283,Z 691.44,A -85,B 0,C 180,E1 1622.211,E2 1622.211} C_VEL
LIN {X 0,Y 587.444,Z 691.44,A -85,B 0,C 180,E1 1628.415,E2 1628.415} C_VEL
LIN {X 0,Y 578.648,Z 691.44,A -85,B 0,C 180,E1 1631.801,E2 1631.801} C_VEL
LIN {X 0,Y 578.553,Z 691.44,A -85,B 0,C 180,E1 1639.123,E2 1639.123} C_VEL
LIN {X 0,Y 578.458,Z 691.44,A -85,B 0,C 180,E1 1645.629,E2 1645.629} C_VEL
LIN {X 0,Y 578.579,Z 691.44,A -85,B 0,C 180,E1 1652.502,E2 1652.502} C_VEL
LIN {X 0,Y 578.467,Z 691.44,A -85,B 0,C 180,E1 1661.609,E2 1661.609} C_VEL
LIN {X 0,Y 578.5,Z 691.44,A -85,B 0,C 180,E1 1670.005,E2 1670.005} C_VEL
LIN {X 0,Y 579.017,Z 693.387,A -85,B 0,C 180,E1 1674.425,E2 1674.425} C_VEL
LIN {X 0,Y 584.255,Z 707.854,A -85,B 0,C 180,E1 1675.004,E2 1675.004} C_VEL
LIN {X 0,Y 584.337,Z 783.354,A -85,B 0,C 180,E1 1676.67,E2 1676.67} C_VEL
LIN {X 0,Y 582.951,Z 846.472,A -85,B 0,C 180,E1 1679.586,E2 1679.586} C_VEL
LIN {X 0,Y 581.183,Z 906.713,A -85,B 0,C 180,E1 1684.113,E2 1684.113} C_VEL
LIN {X 0,Y 579.854,Z 954.534,A -85,B 0,C 180,E1 1689.522,E2 1689.522} C_VEL
LIN {X 0,Y 579.16,Z 988.548,A -85,B 0,C 180,E1 1695.198,E2 1695.198} C_VEL
LIN {X 0,Y 579.069,Z 1010.376,A -85,B 0,C 180,E1 1700.953,E2 1700.953} C_VEL
LIN {X 0,Y 579.433,Z 1020.766,A -85,B 0,C 180,E1 1706.245,E2 1706.245} C_VEL
LIN {X 0,Y 579.345,Z 1022.149,A -85,B 0,C 180,E1 1712.252,E2 1712.252} C_VEL
LIN {X 0,Y 579.188,Z 1010.378,A -85,B 0,C 180,E1 1719.045,E2 1719.045} C_VEL
LIN {X 0,Y 579.469,Z 984.614,A -85,B 0,C 180,E1 1725.571,E2 1725.571} C_VEL
LIN {X 0,Y 580.32,Z 946.182,A -85,B 0,C 180,E1 1731.576,E2 1731.576} C_VEL
LIN {X 0,Y 581.663,Z 894.352,A -85,B 0,C 180,E1 1736.978,E2 1736.978} C_VEL
LIN {X 0,Y 583.368,Z 833.326,A -85,B 0,C 180,E1 1741.154,E2 1741.154} C_VEL
LIN {X 0,Y 584.632,Z 769.889,A -85,B 0,C 180,E1 1743.747,E2 1743.747} C_VEL
LIN {X 0,Y 582.582,Z 699.439,A -85,B 0,C 180,E1 1745.235,E2 1745.235} C_VEL
LIN {X 0,Y 579.282,Z 691.44,A -85,B 0,C 180,E1 1745.702,E2 1745.702} C_VEL
LIN {X 0,Y 578.32,Z 691.44,A -85,B 0,C 180,E1 1754.058,E2 1754.058} C_VEL
LIN {X 0,Y 578.201,Z 691.44,A -85,B 0,C 180,E1 1760.739,E2 1760.739} C_VEL
LIN {X 0,Y 578.615,Z 691.44,A -85,B 0,C 180,E1 1768.474,E2 1768.474} C_VEL
LIN {X 0,Y 578.678,Z 691.44,A -85,B 0,C 180,E1 1776.036,E2 1776.036} C_VEL
LIN {X 0,Y 579.179,Z 691.44,A -85,B 0,C 180,E1 1784.047,E2 1784.047} C_VEL
LIN {X 0,Y 579.099,Z 691.44,A -85,B 0,C 180,E1 1793.24,E2 1793.24} C_VEL
LIN {X 0,Y 578.993,Z 691.44,A -85,B 0,C 180,E1 1800.761,E2 1800.761} C_VEL
LIN {X 0,Y 578.802,Z 691.44,A -85,B 0,C 180,E1 1808.299,E2 1808.299} C_VEL
LIN {X 0,Y 578.646,Z 691.44,A -85,B 0,C 180,E1 1815.989,E2 1815.989} C_VEL
LIN {X 0,Y 578.676,Z 691.44,A -85,B 0,C 180,E1 1822.353,E2 1822.353} C_VEL
LIN {X 0,Y 578.878,Z 692.199,A -85,B 0,C 180,E1 1826.799,E2 1826.799} C_VEL
LIN {X 0,Y 584.376,Z 709.046,A -85,B 0,C 180,E1 1827.45,E2 1827.45} C_VEL
LIN {X 0,Y 583.809,Z 776.552,A -85,B 0,C 180,E1 1829.502,E2 1829.502} C_VEL
LIN {X 0,Y 582.442,Z 839.667,A -85,B 0,C 180,E1 1833.061,E2 1833.061} C_VEL
LIN {X 0,Y 580.998,Z 895.557,A -85,B 0,C 180,E1 1837.974,E2 1837.974} C_VEL
LIN {X 0,Y 580.131,Z 940.469,A -85,B 0,C 180,E1 1843.88,E2 1843.88} C_VEL
LIN {X 0,Y 579.668,Z 971.12,A -85,B 0,C 180,E1 1850.103,E2 1850.103} C_VEL
LIN {X 0,Y 579.475,Z 988.47,A -85,B 0,C 180,E1 1856.557,E2 1856.557} C_VEL
LIN {X 0,Y 579.222,Z 992.841,A -85,B 0,C 180,E1 1862.709,E2 1862.709} C_VEL
LIN {X 0,Y 579.451,Z 984.708,A -85,B 0,C 180,E1 1869.295,E2 1869.295} C_VEL
LIN {X 0,Y 579.607,Z 962.03,A -85,B 0,C 180,E1 1875.984,E2 1875.984} C_VEL
LIN {X 0,Y 580.192,Z 925.457,A -85,B 0,C 180,E1 1882.296,E2 1882.296} C_VEL
LIN {X 0,Y 581.44,Z 875.46,A -85,B 0,C 180,E1 1887.944,E2 1887.944} C_VEL
LIN {X 0,Y 583.066,Z 817.005,A -85,B 0,C 180,E1 1892.331,E2 1892.331} C_VEL
LIN {X 0,Y 584.362,Z 752.85,A -85,B 0,C 180,E1 1895.302,E2 1895.302} C_VEL
LIN {X 0,Y 582.825,Z 699.51,A -85,B 0,C 180,E1 1896.729,E2 1896.729} C_VEL
LIN {X 0,Y 579.659,Z 691.44,A -85,B 0,C 180,E1 1897.144,E2 1897.144} C_VEL
LIN {X 0,Y 578.972,Z 691.44,A -85,B 0,C 180,E1 1906.948,E2 1906.948} C_VEL
LIN {X 0,Y 578.627,Z 691.44,A -85,B 0,C 180,E1 1915.217,E2 1915.217} C_VEL
LIN {X 0,Y 578.619,Z 691.44,A -85,B 0,C 180,E1 1922.526,E2 1922.526} C_VEL
LIN {X 0,Y 578.533,Z 691.44,A -85,B 0,C 180,E1 1931.624,E2 1931.624} C_VEL
LIN {X 0,Y 578.429,Z 691.44,A -85,B 0,C 180,E1 1940.004,E2 1940.004} C_VEL
LIN {X 0,Y 578.669,Z 691.44,A -85,B 0,C 180,E1 1948.467,E2 1948.467} C_VEL
LIN {X 0,Y 578.714,Z 691.44,A -85,B 0,C 180,E1 1956.015,E2 1956.015} C_VEL
LIN {X 0,Y 579.622,Z 691.44,A -85,B 0,C 180,E1 1965.592,E2 1965.592} C_VEL
LIN {X 0,Y 579.363,Z 691.44,A -85,B 0,C 180,E1 1974.731,E2 1974.731} C_VEL
LIN {X 0,Y 579.292,Z 691.44,A -85,B 0,C 180,E1 1982.241,E2 1982.241} C_VEL
LIN {X 0,Y 578.796,Z 691.44,A -85,B 0,C 180,E1 1990.502,E2 1990.502} C_VEL
LIN {X 0,Y 578.648,Z 691.44,A -85,B 0,C 180,E1 1991.801,E2 1991.801} C_VEL
LIN {X 0,Y 571.181,Z 691.44,A -85,B 0,C 180,E1 1995.275,E2 1995.275} C_VEL
LIN {X 0,Y 570.851,Z 691.44,A -85,B 0,C 180,E1 2004.314,E2 2004.314} C_VEL
LIN {X 0,Y 570.387,Z 691.44,A -85,B 0,C 180,E1 2013.059,E2 2013.059} C_VEL
LIN {X 0,Y 570.643,Z 691.44,A -85,B 0,C 180,E1 2020.717,E2 2020.717} C_VEL
LIN {X 0,Y 570.685,Z 691.44,A -85,B 0,C 180,E1 2029.344,E2 2029.344} C_VEL
LIN {X 0,Y 570.721,Z 693.215,A -85,B 0,C 180,E1 2033.824,E2 2033.824} C_VEL
LIN {X 0,Y 577.727,Z 709.32,A -85,B 0,C 180,E1 2034.572,E2 2034.572} C_VEL
LIN {X 0,Y 577.578,Z 783.433,A -85,B 0,C 180,E1 2036.23,E2 2036.23} C_VEL
LIN {X 0,Y 575.818,Z 847.483,A -85,B 0,C 180,E1 2039.233,E2 2039.233} C_VEL
LIN {X 0,Y 573.683,Z 906.341,A -85,B 0,C 180,E1 2043.714,E2 2043.714} C_VEL
LIN {X 0,Y 572.059,Z 955.568,A -85,B 0,C 180,E1 2049.374,E2 2049.374} C_VEL
LIN {X 0,Y 571.3,Z 988.547,A -85,B 0,C 180,E1 2054.989,E2 2054.989} C_VEL
LIN {X 0,Y 571.14,Z 1010.375,A -85,B 0,C 180,E1 2060.826,E2 2060.826} C_VEL
LIN {X 0,Y 571.44,Z 1020.766,A -85,B 0,C 180,E1 2066.193,E2 2066.193} C_VEL
LIN {X 0,Y 571.33,Z 1022.149,A -85,B 0,C 180,E1 2072.283,E2 2072.283} C_VEL
LIN {X 0,Y 571.474,Z 1012.354,A -85,B 0,C 180,E1 2078.398,E2 2078.398} C_VEL
LIN {X 0,Y 571.752,Z 988.549,A -85,B 0,C 180,E1 2084.998,E2 2084.998} C_VEL
LIN {X 0,Y 572.566,Z 949.052,A -85,B 0,C 180,E1 2091.506,E2 2091.506} C_VEL
LIN {X 0,Y 574.177,Z 898.145,A -85,B 0,C 180,E1 2097.018,E2 2097.018} C_VEL
LIN {X 0,Y 576.117,Z 839.493,A -85,B 0,C 180,E1 2101.231,E2 2101.231} C_VEL
LIN {X 0,Y 577.841,Z 774.251,A -85,B 0,C 180,E1 2104.069,E2 2104.069} C_VEL
LIN {X 0,Y 575.933,Z 701.814,A -85,B 0,C 180,E1 2105.668,E2 2105.668} C_VEL
LIN {X 0,Y 571.236,Z 691.44,A -85,B 0,C 180,E1 2106.29,E2 2106.29} C_VEL
LIN {X 0,Y 570.511,Z 691.44,A -85,B 0,C 180,E1 2115.212,E2 2115.212} C_VEL
LIN {X 0,Y 570.386,Z 691.44,A -85,B 0,C 180,E1 2124.242,E2 2124.242} C_VEL
LIN {X 0,Y 570.935,Z 691.44,A -85,B 0,C 180,E1 2134.008,E2 2134.008} C_VEL
LIN {X 0,Y 571.168,Z 691.44,A -85,B 0,C 180,E1 2143.817,E2 2143.817} C_VEL
LIN {X 0,Y 571.113,Z 691.44,A -85,B 0,C 180,E1 2153.145,E2 2153.145} C_VEL
LIN {X 0,Y 570.988,Z 691.44,A -85,B 0,C 180,E1 2160.772,E2 2160.772} C_VEL
LIN {X 0,Y 570.785,Z 691.44,A -85,B 0,C 180,E1 2168.416,E2 2168.416} C_VEL
LIN {X 0,Y 570.63,Z 691.44,A -85,B 0,C 180,E1 2176.22,E2 2176.22} C_VEL
LIN {X 0,Y 570.412,Z 691.44,A -85,B 0,C 180,E1 2183.383,E2 2183.383} C_VEL
LIN {X 0,Y 570.769,Z 692.928,A -85,B 0,C 180,E1 2186.235,E2 2186.235} C_VEL
LIN {X 0,Y 577.816,Z 711.639,A -85,B 0,C 180,E1 2187.047,E2 2187.047} C_VEL
LIN {X 0,Y 576.816,Z 779.338,A -85,B 0,C 180,E1 2189.187,E2 2189.187} C_VEL
LIN {X 0,Y 575.117,Z 842.478,A -85,B 0,C 180,E1 2192.864,E2 2192.864} C_VEL
LIN {X 0,Y 573.365,Z 898.025,A -85,B 0,C 180,E1 2197.902,E2 2197.902} C_VEL
LIN {X 0,Y 572.323,Z 942.993,A -85,B 0,C 180,E1 2204.04,E2 2204.04} C_VEL
LIN {X 0,Y 571.795,Z 973.712,A -85,B 0,C 180,E1 2210.678,E2 2210.678} C_VEL
LIN {X 0,Y 571.388,Z 989.314,A -85,B 0,C 180,E1 2217.012,E2 2217.012} C_VEL
LIN {X 0,Y 571.138,Z 992.318,A -85,B 0,C 180,E1 2223.997,E2 2223.997} C_VEL
LIN {X 0,Y 571.139,Z 982.772,A -85,B 0,C 180,E1 2230.198,E2 2230.198} C_VEL
LIN {X 0,Y 571.444,Z 960.13,A -85,B 0,C 180,E1 2236.613,E2 2236.613} C_VEL
LIN {X 0,Y 572.348,Z 922.784,A -85,B 0,C 180,E1 2242.956,E2 2242.956} C_VEL
LIN {X 0,Y 573.972,Z 873.542,A -85,B 0,C 180,E1 2248.485,E2 2248.485} C_VEL
LIN {X 0,Y 576,Z 814.049,A -85,B 0,C 180,E1 2252.926,E2 2252.926} C_VEL
LIN {X 0,Y 577.728,Z 749.78,A -85,B 0,C 180,E1 2255.843,E2 2255.843} C_VEL
LIN {X 0,Y 576.383,Z 702.368,A -85,B 0,C 180,E1 2257.126,E2 2257.126} C_VEL
LIN {X 0,Y 571.64,Z 691.44,A -85,B 0,C 180,E1 2257.771,E2 2257.771} C_VEL
LIN {X 0,Y 571.283,Z 691.44,A -85,B 0,C 180,E1 2266.197,E2 2266.197} C_VEL
LIN {X 0,Y 570.91,Z 691.44,A -85,B 0,C 180,E1 2274.332,E2 2274.332} C_VEL
LIN {X 0,Y 570.413,Z 691.44,A -85,B 0,C 180,E1 2283.077,E2 2283.077} C_VEL
LIN {X 0,Y 570.694,Z 691.44,A -85,B 0,C 180,E1 2290.731,E2 2290.731} C_VEL
LIN {X 0,Y 570.65,Z 691.44,A -85,B 0,C 180,E1 2299.345,E2 2299.345} C_VEL
LIN {X 0,Y 570.606,Z 691.44,A -85,B 0,C 180,E1 2308.76,E2 2308.76} C_VEL
LIN {X 0,Y 570.447,Z 691.44,A -85,B 0,C 180,E1 2316.611,E2 2316.611} C_VEL
LIN {X 0,Y 571.596,Z 691.44,A -85,B 0,C 180,E1 2325.715,E2 2325.715} C_VEL
LIN {X 0,Y 571.263,Z 691.44,A -85,B 0,C 180,E1 2335.012,E2 2335.012} C_VEL
LIN {X 0,Y 571.271,Z 691.44,A -85,B 0,C 180,E1 2342.273,E2 2342.273} C_VEL
LIN {X 0,Y 570.969,Z 691.44,A -85,B 0,C 180,E1 2349.934,E2 2349.934} C_VEL
LIN {X 0,Y 571.181,Z 691.44,A -85,B 0,C 180,E1 2355.275,E2 2355.275} C_VEL
LIN {X 0,Y 562.566,Z 691.44,A -85,B 0,C 180,E1 2358.76,E2 2358.76} C_VEL
LIN {X 0,Y 562.373,Z 691.44,A -85,B 0,C 180,E1 2366.418,E2 2366.418} C_VEL
LIN {X 0,Y 562.263,Z 691.44,A -85,B 0,C 180,E1 2373.568,E2 2373.568} C_VEL
LIN {X 0,Y 562.334,Z 691.44,A -85,B 0,C 180,E1 2382.084,E2 2382.084} C_VEL
LIN {X 0,Y 562.314,Z 691.44,A -85,B 0,C 180,E1 2390.637,E2 2390.637} C_VEL
LIN {X 0,Y 562.467,Z 692.61,A -85,B 0,C 180,E1 2393.198,E2 2393.198} C_VEL
LIN {X 0,Y 571.261,Z 712.961,A -85,B 0,C 180,E1 2394.164,E2 2394.164} C_VEL
LIN {X 0,Y 570.841,Z 785.484,A -85,B 0,C 180,E1 2395.849,E2 2395.849} C_VEL
LIN {X 0,Y 568.708,Z 848.629,A -85,B 0,C 180,E1 2398.881,E2 2398.881} C_VEL
LIN {X 0,Y 566.139,Z 908.341,A -85,B 0,C 180,E1 2403.535,E2 2403.535} C_VEL
LIN {X 0,Y 564.323,Z 955.9,A -85,B 0,C 180,E1 2409.125,E2 2409.125} C_VEL
LIN {X 0,Y 563.284,Z 990.328,A -85,B 0,C 180,E1 2415.17,E2 2415.17} C_VEL
LIN {X 0,Y 563.196,Z 1010.375,A -85,B 0,C 180,E1 2420.695,E2 2420.695} C_VEL
LIN {X 0,Y 563.471,Z 1020.766,A -85,B 0,C 180,E1 2426.139,E2 2426.139} C_VEL
LIN {X 0,Y 563.315,Z 1022.149,A -85,B 0,C 180,E1 2432.316,E2 2432.316} C_VEL
LIN {X 0,Y 563.418,Z 1012.355,A -85,B 0,C 180,E1 2438.519,E2 2438.519} C_VEL
LIN {X 0,Y 563.77,Z 988.548,A -85,B 0,C 180,E1 2445.216,E2 2445.216} C_VEL
LIN {X 0,Y 564.791,Z 950.028,A -85,B 0,C 180,E1 2451.68,E2 2451.68} C_VEL
LIN {X 0,Y 566.707,Z 899.297,A -85,B 0,C 180,E1 2457.296,E2 2457.296} C_VEL
LIN {X 0,Y 569.067,Z 840.634,A -85,B 0,C 180,E1 2461.595,E2 2461.595} C_VEL
LIN {X 0,Y 571.101,Z 775.946,A -85,B 0,C 180,E1 2464.468,E2 2464.468} C_VEL
LIN {X 0,Y 569.695,Z 705.561,A -85,B 0,C 180,E1 2466.062,E2 2466.062} C_VEL
LIN {X 0,Y 563.148,Z 691.44,A -85,B 0,C 180,E1 2466.947,E2 2466.947} C_VEL
LIN {X 0,Y 562.834,Z 691.44,A -85,B 0,C 180,E1 2477.858,E2 2477.858} C_VEL
LIN {X 0,Y 562.569,Z 691.44,A -85,B 0,C 180,E1 2488.287,E2 2488.287} C_VEL
LIN {X 0,Y 562.326,Z 691.44,A -85,B 0,C 180,E1 2496.983,E2 2496.983} C_VEL
LIN {X 0,Y 562.829,Z 691.44,A -85,B 0,C 180,E1 2505.174,E2 2505.174} C_VEL
LIN {X 0,Y 563.122,Z 691.44,A -85,B 0,C 180,E1 2513.048,E2 2513.048} C_VEL
LIN {X 0,Y 562.989,Z 691.44,A -85,B 0,C 180,E1 2520.783,E2 2520.783} C_VEL
LIN {X 0,Y 562.765,Z 691.44,A -85,B 0,C 180,E1 2528.537,E2 2528.537} C_VEL
LIN {X 0,Y 562.64,Z 691.44,A -85,B 0,C 180,E1 2536.759,E2 2536.759} C_VEL
LIN {X 0,Y 562.416,Z 691.44,A -85,B 0,C 180,E1 2545.319,E2 2545.319} C_VEL
LIN {X 0,Y 565.479,Z 698.691,A -85,B 0,C 180,E1 2545.938,E2 2545.938} C_VEL
LIN {X 0,Y 571.241,Z 714.152,A -85,B 0,C 180,E1 2546.637,E2 2546.637} C_VEL
LIN {X 0,Y 569.836,Z 782.848,A -85,B 0,C 180,E1 2548.9,E2 2548.9} C_VEL
LIN {X 0,Y 567.782,Z 845.054,A -85,B 0,C 180,E1 2552.655,E2 2552.655} C_VEL
LIN {X 0,Y 565.7,Z 899.678,A -85,B 0,C 180,E1 2557.75,E2 2557.75} C_VEL
LIN {X 0,Y 564.421,Z 943.699,A -85,B 0,C 180,E1 2563.904,E2 2563.904} C_VEL
LIN {X 0,Y 563.777,Z 974.554,A -85,B 0,C 180,E1 2570.76,E2 2570.76} C_VEL
LIN {X 0,Y 563.307,Z 989.884,A -85,B 0,C 180,E1 2577.324,E2 2577.324} C_VEL
LIN {X 0,Y 563.061,Z 991.991,A -85,B 0,C 180,E1 2584.525,E2 2584.525} C_VEL
LIN {X 0,Y 562.988,Z 981.705,A -85,B 0,C 180,E1 2590.75,E2 2590.75} C_VEL
LIN {X 0,Y 563.457,Z 960.397,A -85,B 0,C 180,E1 2596.766,E2 2596.766} C_VEL
LIN {X 0,Y 564.546,Z 924.275,A -85,B 0,C 180,E1 2603.052,E2 2603.052} C_VEL
LIN {X 0,Y 566.492,Z 874.715,A -85,B 0,C 180,E1 2608.753,E2 2608.753} C_VEL
LIN {X 0,Y 568.901,Z 815.734,A -85,B 0,C 180,E1 2613.25,E2 2613.25} C_VEL
LIN {X 0,Y 570.976,Z 751.957,A -85,B 0,C 180,E1 2616.222,E2 2616.222} C_VEL
LIN {X 0,Y 570.011,Z 705.626,A -85,B 0,C 180,E1 2617.522,E2 2617.522} C_VEL
LIN {X 0,Y 563.603,Z 691.44,A -85,B 0,C 180,E1 2618.271,E2 2618.271} C_VEL
LIN {X 0,Y 562.981,Z 691.44,A -85,B 0,C 180,E1 2626.904,E2 2626.904} C_VEL
LIN {X 0,Y 562.578,Z 691.44,A -85,B 0,C 180,E1 2635.372,E2 2635.372} C_VEL
LIN {X 0,Y 562.298,Z 691.44,A -85,B 0,C 180,E1 2643.592,E2 2643.592} C_VEL
LIN {X 0,Y 562.374,Z 691.44,A -85,B 0,C 180,E1 2652.096,E2 2652.096} C_VEL
LIN {X 0,Y 562.343,Z 691.44,A -85,B 0,C 180,E1 2660.276,E2 2660.276} C_VEL
LIN {X 0,Y 562.624,Z 691.44,A -85,B 0,C 180,E1 2668.266,E2 2668.266} C_VEL
LIN {X 0,Y 562.321,Z 691.44,A -85,B 0,C 180,E1 2676.96,E2 2676.96} C_VEL
LIN {X 0,Y 563.511,Z 691.44,A -85,B 0,C 180,E1 2686.761,E2 2686.761} C_VEL
LIN {X 0,Y 562.94,Z 691.44,A -85,B 0,C 180,E1 2696.126,E2 2696.126} C_VEL
LIN {X 0,Y 562.822,Z 691.44,A -85,B 0,C 180,E1 2703.853,E2 2703.853} C_VEL
LIN {X 0,Y 562.649,Z 691.44,A -85,B 0,C 180,E1 2711.656,E2 2711.656} C_VEL
LIN {X 0,Y 562.566,Z 691.44,A -85,B 0,C 180,E1 2718.76,E2 2718.76} C_VEL
LIN {X 0,Y 554.858,Z 691.44,A -85,B 0,C 180,E1 2722.306,E2 2722.306} C_VEL
LIN {X 0,Y 554.553,Z 691.44,A -85,B 0,C 180,E1 2732.226,E2 2732.226} C_VEL
LIN {X 0,Y 554.463,Z 691.44,A -85,B 0,C 180,E1 2741.176,E2 2741.176} C_VEL
LIN {X 0,Y 554.436,Z 691.44,A -85,B 0,C 180,E1 2749.966,E2 2749.966} C_VEL
LIN {X 0,Y 554.496,Z 693.381,A -85,B 0,C 180,E1 2752.591,E2 2752.591} C_VEL
LIN {X 0,Y 564.774,Z 714.733,A -85,B 0,C 180,E1 2753.715,E2 2753.715} C_VEL
LIN {X 0,Y 564.145,Z 786.079,A -85,B 0,C 180,E1 2755.408,E2 2755.408} C_VEL
LIN {X 0,Y 561.65,Z 849.487,A -85,B 0,C 180,E1 2758.503,E2 2758.503} C_VEL
LIN {X 0,Y 558.757,Z 908.408,A -85,B 0,C 180,E1 2763.164,E2 2763.164} C_VEL
LIN {X 0,Y 556.515,Z 957.348,A -85,B 0,C 180,E1 2769.028,E2 2769.028} C_VEL
LIN {X 0,Y 555.389,Z 990.33,A -85,B 0,C 180,E1 2774.954,E2 2774.954} C_VEL
LIN {X 0,Y 555.266,Z 1010.374,A -85,B 0,C 180,E1 2780.561,E2 2780.561} C_VEL
LIN {X 0,Y 555.477,Z 1020.766,A -85,B 0,C 180,E1 2786.083,E2 2786.083} C_VEL
LIN {X 0,Y 555.301,Z 1022.15,A -85,B 0,C 180,E1 2792.349,E2 2792.349} C_VEL
LIN {X 0,Y 555.365,Z 1012.355,A -85,B 0,C 180,E1 2798.644,E2 2798.644} C_VEL
LIN {X 0,Y 555.773,Z 988.547,A -85,B 0,C 180,E1 2805.44,E2 2805.44} C_VEL
LIN {X 0,Y 557.026,Z 950.549,A -85,B 0,C 180,E1 2811.924,E2 2811.924} C_VEL
LIN {X 0,Y 559.288,Z 899.883,A -85,B 0,C 180,E1 2817.633,E2 2817.633} C_VEL
LIN {X 0,Y 562.028,Z 841.889,A -85,B 0,C 180,E1 2821.962,E2 2821.962} C_VEL
LIN {X 0,Y 564.383,Z 777.522,A -85,B 0,C 180,E1 2824.881,E2 2824.881} C_VEL
LIN {X 0,Y 563.371,Z 708.807,A -85,B 0,C 180,E1 2826.482,E2 2826.482} C_VEL
LIN {X 0,Y 555.102,Z 691.44,A -85,B 0,C 180,E1 2827.542,E2 2827.542} C_VEL
LIN {X 0,Y 554.813,Z 691.44,A -85,B 0,C 180,E1 2837.954,E2 2837.954} C_VEL
LIN {X 0,Y 554.596,Z 691.44,A -85,B 0,C 180,E1 2847.777,E2 2847.777} C_VEL
LIN {X 0,Y 554.382,Z 691.44,A -85,B 0,C 180,E1 2856.634,E2 2856.634} C_VEL
LIN {X 0,Y 554.839,Z 691.44,A -85,B 0,C 180,E1 2864.956,E2 2864.956} C_VEL
LIN {X 0,Y 555.134,Z 691.44,A -85,B 0,C 180,E1 2872.947,E2 2872.947} C_VEL
LIN {X 0,Y 554.984,Z 691.44,A -85,B 0,C 180,E1 2880.794,E2 2880.794} C_VEL
LIN {X 0,Y 554.777,Z 691.44,A -85,B 0,C 180,E1 2888.661,E2 2888.661} C_VEL
LIN {X 0,Y 554.637,Z 691.44,A -85,B 0,C 180,E1 2896.701,E2 2896.701} C_VEL
LIN {X 0,Y 554.42,Z 692.37,A -85,B 0,C 180,E1 2905.002,E2 2905.002} C_VEL
LIN {X 0,Y 564.694,Z 716.266,A -85,B 0,C 180,E1 2906.213,E2 2906.213} C_VEL
LIN {X 0,Y 562.955,Z 785.328,A -85,B 0,C 180,E1 2908.561,E2 2908.561} C_VEL
LIN {X 0,Y 560.468,Z 847.254,A -85,B 0,C 180,E1 2912.412,E2 2912.412} C_VEL
LIN {X 0,Y 558.032,Z 901.189,A -85,B 0,C 180,E1 2917.576,E2 2917.576} C_VEL
LIN {X 0,Y 556.516,Z 944.203,A -85,B 0,C 180,E1 2923.727,E2 2923.727} C_VEL
LIN {X 0,Y 555.834,Z 974.69,A -85,B 0,C 180,E1 2930.637,E2 2930.637} C_VEL
LIN {X 0,Y 555.194,Z 990.514,A -85,B 0,C 180,E1 2937.791,E2 2937.791} C_VEL
LIN {X 0,Y 555.047,Z 991.756,A -85,B 0,C 180,E1 2944.926,E2 2944.926} C_VEL
LIN {X 0,Y 554.919,Z 981.091,A -85,B 0,C 180,E1 2951.125,E2 2951.125} C_VEL
LIN {X 0,Y 555.422,Z 958.684,A -85,B 0,C 180,E1 2957.374,E2 2957.374} C_VEL
LIN {X 0,Y 556.776,Z 922.772,A -85,B 0,C 180,E1 2963.575,E2 2963.575} C_VEL
LIN {X 0,Y 559.084,Z 873.823,A -85,B 0,C 180,E1 2969.223,E2 2969.223} C_VEL
LIN {X 0,Y 561.915,Z 815.82,A -85,B 0,C 180,E1 2973.678,E2 2973.678} C_VEL
LIN {X 0,Y 564.276,Z 752.698,A -85,B 0,C 180,E1 2976.661,E2 2976.661} C_VEL
LIN {X 0,Y 563.411,Z 708.477,A -85,B 0,C 180,E1 2977.951,E2 2977.951} C_VEL
LIN {X 0,Y 555.288,Z 691.44,A -85,B 0,C 180,E1 2979.042,E2 2979.042} C_VEL
LIN {X 0,Y 555.083,Z 691.44,A -85,B 0,C 180,E1 2986.683,E2 2986.683} C_VEL
LIN {X 0,Y 554.672,Z 691.44,A -85,B 0,C 180,E1 2995.093,E2 2995.093} C_VEL
LIN {X 0,Y 554.339,Z 691.44,A -85,B 0,C 180,E1 3003.397,E2 3003.397} C_VEL
LIN {X 0,Y 554.379,Z 691.44,A -85,B 0,C 180,E1 3012.12,E2 3012.12} C_VEL
LIN {X 0,Y 554.391,Z 691.44,A -85,B 0,C 180,E1 3019.966,E2 3019.966} C_VEL
LIN {X 0,Y 554.649,Z 691.44,A -85,B 0,C 180,E1 3027.755,E2 3027.755} C_VEL
LIN {X 0,Y 554.385,Z 691.44,A -85,B 0,C 180,E1 3036.611,E2 3036.611} C_VEL
LIN {X 0,Y 555.49,Z 691.44,A -85,B 0,C 180,E1 3046.566,E2 3046.566} C_VEL
LIN {X 0,Y 554.961,Z 691.44,A -85,B 0,C 180,E1 3056.071,E2 3056.071} C_VEL
LIN {X 0,Y 554.841,Z 691.44,A -85,B 0,C 180,E1 3063.909,E2 3063.909} C_VEL
LIN {X 0,Y 554.65,Z 691.44,A -85,B 0,C 180,E1 3071.827,E2 3071.827} C_VEL
LIN {X 0,Y 554.605,Z 691.44,A -85,B 0,C 180,E1 3079.983,E2 3079.983} C_VEL
LIN {X 0,Y 554.858,Z 691.44,A -85,B 0,C 180,E1 3082.306,E2 3082.306} C_VEL
LIN {X 0,Y 546.458,Z 691.44,A -85,B 0,C 180,E1 3085.891,E2 3085.891} C_VEL
LIN {X 0,Y 546.405,Z 691.44,A -85,B 0,C 180,E1 3092.766,E2 3092.766} C_VEL
LIN {X 0,Y 546.516,Z 691.44,A -85,B 0,C 180,E1 3100.703,E2 3100.703} C_VEL
LIN {X 0,Y 546.485,Z 691.44,A -85,B 0,C 180,E1 3109.748,E2 3109.748} C_VEL
LIN {X 0,Y 546.468,Z 693.431,A -85,B 0,C 180,E1 3111.945,E2 3111.945} C_VEL
LIN {X 0,Y 558.381,Z 718.426,A -85,B 0,C 180,E1 3113.29,E2 3113.29} C_VEL
LIN {X 0,Y 557.451,Z 788.05,A -85,B 0,C 180,E1 3115.004,E2 3115.004} C_VEL
LIN {X 0,Y 554.489,Z 852.327,A -85,B 0,C 180,E1 3118.241,E2 3118.241} C_VEL
LIN {X 0,Y 551.224,Z 910.444,A -85,B 0,C 180,E1 3122.982,E2 3122.982} C_VEL
LIN {X 0,Y 548.837,Z 957.348,A -85,B 0,C 180,E1 3128.72,E2 3128.72} C_VEL
LIN {X 0,Y 547.413,Z 991.402,A -85,B 0,C 180,E1 3134.98,E2 3134.98} C_VEL
LIN {X 0,Y 546.987,Z 1012.354,A -85,B 0,C 180,E1 3141.222,E2 3141.222} C_VEL
LIN {X 0,Y 546.921,Z 1022.149,A -85,B 0,C 180,E1 3147.614,E2 3147.614} C_VEL
LIN {X 0,Y 547.032,Z 1020.768,A -85,B 0,C 180,E1 3153.977,E2 3153.977} C_VEL
LIN {X 0,Y 546.926,Z 1008.898,A -85,B 0,C 180,E1 3160.101,E2 3160.101} C_VEL
LIN {X 0,Y 547.651,Z 984.619,A -85,B 0,C 180,E1 3166.501,E2 3166.501} C_VEL
LIN {X 0,Y 549.322,Z 947.327,A -85,B 0,C 180,E1 3172.707,E2 3172.707} C_VEL
LIN {X 0,Y 552.156,Z 895.461,A -85,B 0,C 180,E1 3178.448,E2 3178.448} C_VEL
LIN {X 0,Y 555.467,Z 835.315,A -85,B 0,C 180,E1 3182.788,E2 3182.788} C_VEL
LIN {X 0,Y 558.06,Z 771.915,A -85,B 0,C 180,E1 3185.528,E2 3185.528} C_VEL
LIN {X 0,Y 556.765,Z 711.26,A -85,B 0,C 180,E1 3186.947,E2 3186.947} C_VEL
LIN {X 0,Y 547,Z 691.44,A -85,B 0,C 180,E1 3188.242,E2 3188.242} C_VEL
LIN {X 0,Y 546.75,Z 691.44,A -85,B 0,C 180,E1 3197.353,E2 3197.353} C_VEL
LIN {X 0,Y 546.588,Z 691.44,A -85,B 0,C 180,E1 3207.867,E2 3207.867} C_VEL
LIN {X 0,Y 546.472,Z 691.44,A -85,B 0,C 180,E1 3216.275,E2 3216.275} C_VEL
LIN {X 0,Y 546.841,Z 691.44,A -85,B 0,C 180,E1 3224.73,E2 3224.73} C_VEL
LIN {X 0,Y 547.134,Z 691.44,A -85,B 0,C 180,E1 3232.843,E2 3232.843} C_VEL
LIN {X 0,Y 546.994,Z 691.44,A -85,B 0,C 180,E1 3240.805,E2 3240.805} C_VEL
LIN {X 0,Y 546.762,Z 691.44,A -85,B 0,C 180,E1 3248.789,E2 3248.789} C_VEL
LIN {X 0,Y 546.657,Z 691.44,A -85,B 0,C 180,E1 3256.952,E2 3256.952} C_VEL
LIN {X 0,Y 546.578,Z 693.333,A -85,B 0,C 180,E1 3264.397,E2 3264.397} C_VEL
LIN {X 0,Y 558.201,Z 718.701,A -85,B 0,C 180,E1 3265.787,E2 3265.787} C_VEL
LIN {X 0,Y 556.091,Z 787.172,A -85,B 0,C 180,E1 3268.189,E2 3268.189} C_VEL
LIN {X 0,Y 553.227,Z 848.029,A -85,B 0,C 180,E1 3272.049,E2 3272.049} C_VEL
LIN {X 0,Y 550.41,Z 901.639,A -85,B 0,C 180,E1 3277.271,E2 3277.271} C_VEL
LIN {X 0,Y 548.617,Z 945.164,A -85,B 0,C 180,E1 3283.63,E2 3283.63} C_VEL
LIN {X 0,Y 547.836,Z 974.603,A -85,B 0,C 180,E1 3290.443,E2 3290.443} C_VEL
LIN {X 0,Y 547.198,Z 990.543,A -85,B 0,C 180,E1 3297.754,E2 3297.754} C_VEL
LIN {X 0,Y 547.002,Z 992.039,A -85,B 0,C 180,E1 3304.531,E2 3304.531} C_VEL
LIN {X 0,Y 547,Z 982.114,A -85,B 0,C 180,E1 3310.841,E2 3310.841} C_VEL
LIN {X 0,Y 547.5,Z 960.484,A -85,B 0,C 180,E1 3317.189,E2 3317.189} C_VEL
LIN {X 0,Y 549.005,Z 924.213,A -85,B 0,C 180,E1 3323.69,E2 3323.69} C_VEL
LIN {X 0,Y 551.622,Z 875.004,A -85,B 0,C 180,E1 3329.508,E2 3329.508} C_VEL
LIN {X 0,Y 554.93,Z 815.934,A -85,B 0,C 180,E1 3334.117,E2 3334.117} C_VEL
LIN {X 0,Y 557.662,Z 752.874,A -85,B 0,C 180,E1 3337.126,E2 3337.126} C_VEL
LIN {X 0,Y 557.026,Z 711.419,A -85,B 0,C 180,E1 3338.375,E2 3338.375} C_VEL
LIN {X 0,Y 547.085,Z 691.44,A -85,B 0,C 180,E1 3339.707,E2 3339.707} C_VEL
LIN {X 0,Y 546.637,Z 691.44,A -85,B 0,C 180,E1 3348.619,E2 3348.619} C_VEL
LIN {X 0,Y 546.47,Z 691.44,A -85,B 0,C 180,E1 3357.273,E2 3357.273} C_VEL
LIN {X 0,Y 546.159,Z 691.44,A -85,B 0,C 180,E1 3364.955,E2 3364.955} C_VEL
LIN {X 0,Y 546.308,Z 691.44,A -85,B 0,C 180,E1 3372.89,E2 3372.89} C_VEL
LIN {X 0,Y 546.426,Z 691.44,A -85,B 0,C 180,E1 3379.797,E2 3379.797} C_VEL
LIN {X 0,Y 546.452,Z 691.44,A -85,B 0,C 180,E1 3389.084,E2 3389.084} C_VEL
LIN {X 0,Y 546.488,Z 691.44,A -85,B 0,C 180,E1 3396.252,E2 3396.252} C_VEL
LIN {X 0,Y 547.502,Z 691.44,A -85,B 0,C 180,E1 3406.366,E2 3406.366} C_VEL
LIN {X 0,Y 546.967,Z 691.44,A -85,B 0,C 180,E1 3416.013,E2 3416.013} C_VEL
LIN {X 0,Y 546.833,Z 691.44,A -85,B 0,C 180,E1 3423.966,E2 3423.966} C_VEL
LIN {X 0,Y 546.653,Z 691.44,A -85,B 0,C 180,E1 3432.002,E2 3432.002} C_VEL
LIN {X 0,Y 546.623,Z 691.44,A -85,B 0,C 180,E1 3440.287,E2 3440.287} C_VEL
LIN {X 0,Y 546.458,Z 691.44,A -85,B 0,C 180,E1 3445.891,E2 3445.891} C_VEL
LIN {X 0,Y 538.574,Z 691.44,A -85,B 0,C 180,E1 3449.543,E2 3449.543} C_VEL
LIN {X 0,Y 538.512,Z 691.44,A -85,B 0,C 180,E1 3459.321,E2 3459.321} C_VEL
LIN {X 0,Y 538.566,Z 691.44,A -85,B 0,C 180,E1 3468.532,E2 3468.532} C_VEL
LIN {X 0,Y 538.418,Z 692.94,A -85,B 0,C 180,E1 3471.264,E2 3471.264} C_VEL
LIN {X 0,Y 552,Z 722.015,A -85,B 0,C 180,E1 3472.852,E2 3472.852} C_VEL
LIN {X 0,Y 550.71,Z 790.8,A -85,B 0,C 180,E1 3474.628,E2 3474.628} C_VEL
LIN {X 0,Y 547.42,Z 853.766,A -85,B 0,C 180,E1 3477.882,E2 3477.882} C_VEL
LIN {X 0,Y 543.745,Z 911.652,A -85,B 0,C 180,E1 3482.709,E2 3482.709} C_VEL
LIN {X 0,Y 541.028,Z 958.7,A -85,B 0,C 180,E1 3488.613,E2 3488.613} C_VEL
LIN {X 0,Y 539.469,Z 992.094,A -85,B 0,C 180,E1 3494.917,E2 3494.917} C_VEL
LIN {X 0,Y 539.036,Z 1012.354,A -85,B 0,C 180,E1 3501.092,E2 3501.092} C_VEL
LIN {X 0,Y 538.93,Z 1022.149,A -85,B 0,C 180,E1 3507.579,E2 3507.579} C_VEL
LIN {X 0,Y 539.021,Z 1020.768,A -85,B 0,C 180,E1 3514.036,E2 3514.036} C_VEL
LIN {X 0,Y 538.938,Z 1009.316,A -85,B 0,C 180,E1 3520.104,E2 3520.104} C_VEL
LIN {X 0,Y 539.747,Z 986.59,A -85,B 0,C 180,E1 3526.33,E2 3526.33} C_VEL
LIN {X 0,Y 541.509,Z 950.128,A -85,B 0,C 180,E1 3532.649,E2 3532.649} C_VEL
LIN {X 0,Y 544.583,Z 899.176,A -85,B 0,C 180,E1 3538.515,E2 3538.515} C_VEL
LIN {X 0,Y 548.311,Z 839.739,A -85,B 0,C 180,E1 3542.996,E2 3542.996} C_VEL
LIN {X 0,Y 551.381,Z 775.255,A -85,B 0,C 180,E1 3545.912,E2 3545.912} C_VEL
LIN {X 0,Y 550.521,Z 714.599,A -85,B 0,C 180,E1 3547.384,E2 3547.384} C_VEL
LIN {X 0,Y 538.929,Z 691.44,A -85,B 0,C 180,E1 3548.862,E2 3548.862} C_VEL
LIN {X 0,Y 538.543,Z 691.44,A -85,B 0,C 180,E1 3558.563,E2 3558.563} C_VEL
LIN {X 0,Y 538.452,Z 691.44,A -85,B 0,C 180,E1 3568.599,E2 3568.599} C_VEL
LIN {X 0,Y 538.46,Z 691.44,A -85,B 0,C 180,E1 3576.344,E2 3576.344} C_VEL
LIN {X 0,Y 538.838,Z 691.44,A -85,B 0,C 180,E1 3584.498,E2 3584.498} C_VEL
LIN {X 0,Y 539.13,Z 691.44,A -85,B 0,C 180,E1 3592.736,E2 3592.736} C_VEL
LIN {X 0,Y 538.89,Z 691.44,A -85,B 0,C 180,E1 3601.344,E2 3601.344} C_VEL
LIN {X 0,Y 538.769,Z 691.44,A -85,B 0,C 180,E1 3608.92,E2 3608.92} C_VEL
LIN {X 0,Y 538.655,Z 691.44,A -85,B 0,C 180,E1 3617.212,E2 3617.212} C_VEL
LIN {X 0,Y 538.559,Z 692.986,A -85,B 0,C 180,E1 3623.732,E2 3623.732} C_VEL
LIN {X 0,Y 551.653,Z 722.302,A -85,B 0,C 180,E1 3625.377,E2 3625.377} C_VEL
LIN {X 0,Y 549.14,Z 790.472,A -85,B 0,C 180,E1 3627.883,E2 3627.883} C_VEL
LIN {X 0,Y 545.769,Z 852.727,A -85,B 0,C 180,E1 3631.995,E2 3631.995} C_VEL
LIN {X 0,Y 542.609,Z 906.398,A -85,B 0,C 180,E1 3637.487,E2 3637.487} C_VEL
LIN {X 0,Y 540.722,Z 949.014,A -85,B 0,C 180,E1 3644.092,E2 3644.092} C_VEL
LIN {X 0,Y 539.628,Z 977.394,A -85,B 0,C 180,E1 3651.176,E2 3651.176} C_VEL
LIN {X 0,Y 539.123,Z 990.818,A -85,B 0,C 180,E1 3657.948,E2 3657.948} C_VEL
LIN {X 0,Y 538.973,Z 992.322,A -85,B 0,C 180,E1 3664.124,E2 3664.124} C_VEL
LIN {X 0,Y 539.087,Z 983.126,A -85,B 0,C 180,E1 3670.547,E2 3670.547} C_VEL
LIN {X 0,Y 539.605,Z 962.253,A -85,B 0,C 180,E1 3676.998,E2 3676.998} C_VEL
LIN {X 0,Y 541.191,Z 927.247,A -85,B 0,C 180,E1 3683.561,E2 3683.561} C_VEL
LIN {X 0,Y 544.11,Z 878.167,A -85,B 0,C 180,E1 3689.601,E2 3689.601} C_VEL
LIN {X 0,Y 547.81,Z 819.194,A -85,B 0,C 180,E1 3694.37,E2 3694.37} C_VEL
LIN {X 0,Y 550.89,Z 756.962,A -85,B 0,C 180,E1 3697.469,E2 3697.469} C_VEL
LIN {X 0,Y 550.319,Z 714.039,A -85,B 0,C 180,E1 3698.833,E2 3698.833} C_VEL
LIN {X 0,Y 538.979,Z 691.44,A -85,B 0,C 180,E1 3700.17,E2 3700.17} C_VEL
LIN {X 0,Y 538.611,Z 691.44,A -85,B 0,C 180,E1 3708.907,E2 3708.907} C_VEL
LIN {X 0,Y 538.467,Z 691.44,A -85,B 0,C 180,E1 3717.712,E2 3717.712} C_VEL
LIN {X 0,Y 538.27,Z 691.44,A -85,B 0,C 180,E1 3726.541,E2 3726.541} C_VEL
LIN {X 0,Y 538.559,Z 691.44,A -85,B 0,C 180,E1 3736.344,E2 3736.344} C_VEL
LIN {X 0,Y 538.572,Z 691.44,A -85,B 0,C 180,E1 3746.67,E2 3746.67} C_VEL
LIN {X 0,Y 538.477,Z 691.44,A -85,B 0,C 180,E1 3756.342,E2 3756.342} C_VEL
LIN {X 0,Y 539.473,Z 691.44,A -85,B 0,C 180,E1 3766.16,E2 3766.16} C_VEL
LIN {X 0,Y 538.973,Z 691.44,A -85,B 0,C 180,E1 3775.954,E2 3775.954} C_VEL
LIN {X 0,Y 538.842,Z 691.44,A -85,B 0,C 180,E1 3784.025,E2 3784.025} C_VEL
LIN {X 0,Y 538.661,Z 691.44,A -85,B 0,C 180,E1 3792.183,E2 3792.183} C_VEL
LIN {X 0,Y 538.658,Z 691.44,A -85,B 0,C 180,E1 3800.601,E2 3800.601} C_VEL
LIN {X 0,Y 538.574,Z 691.44,A -85,B 0,C 180,E1 3809.543,E2 3809.543} C_VEL
LIN {X 0,Y 530.211,Z 691.44,A -85,B 0,C 180,E1 3813.26,E2 3813.26} C_VEL
LIN {X 0,Y 530.251,Z 691.44,A -85,B 0,C 180,E1 3822.232,E2 3822.232} C_VEL
LIN {X 0,Y 530.493,Z 693.1,A -85,B 0,C 180,E1 3830.576,E2 3830.576} C_VEL
LIN {X 0,Y 545.648,Z 724.795,A -85,B 0,C 180,E1 3832.39,E2 3832.39} C_VEL
LIN {X 0,Y 544.054,Z 792.219,A -85,B 0,C 180,E1 3834.191,E2 3834.191} C_VEL
LIN {X 0,Y 540.339,Z 856.059,A -85,B 0,C 180,E1 3837.571,E2 3837.571} C_VEL
LIN {X 0,Y 536.166,Z 914.308,A -85,B 0,C 180,E1 3842.579,E2 3842.579} C_VEL
LIN {X 0,Y 533.039,Z 961.392,A -85,B 0,C 180,E1 3848.715,E2 3848.715} C_VEL
LIN {X 0,Y 531.601,Z 992.094,A -85,B 0,C 180,E1 3854.688,E2 3854.688} C_VEL
LIN {X 0,Y 531.089,Z 1012.354,A -85,B 0,C 180,E1 3860.957,E2 3860.957} C_VEL
LIN {X 0,Y 530.937,Z 1022.15,A -85,B 0,C 180,E1 3867.542,E2 3867.542} C_VEL
LIN {X 0,Y 531.012,Z 1020.768,A -85,B 0,C 180,E1 3874.097,E2 3874.097} C_VEL
LIN {X 0,Y 530.975,Z 1009.531,A -85,B 0,C 180,E1 3880.179,E2 3880.179} C_VEL
LIN {X 0,Y 531.846,Z 985.509,A -85,B 0,C 180,E1 3886.814,E2 3886.814} C_VEL
LIN {X 0,Y 533.941,Z 948.547,A -85,B 0,C 180,E1 3893.226,E2 3893.226} C_VEL
LIN {X 0,Y 537.453,Z 897.054,A -85,B 0,C 180,E1 3899.141,E2 3899.141} C_VEL
LIN {X 0,Y 541.628,Z 837.002,A -85,B 0,C 180,E1 3903.629,E2 3903.629} C_VEL
LIN {X 0,Y 544.972,Z 773.384,A -85,B 0,C 180,E1 3906.47,E2 3906.47} C_VEL
LIN {X 0,Y 544.3,Z 717.782,A -85,B 0,C 180,E1 3907.834,E2 3907.834} C_VEL
LIN {X 0,Y 530.742,Z 691.44,A -85,B 0,C 180,E1 3909.66,E2 3909.66} C_VEL
LIN {X 0,Y 530.36,Z 691.44,A -85,B 0,C 180,E1 3919.312,E2 3919.312} C_VEL
LIN {X 0,Y 530.419,Z 691.44,A -85,B 0,C 180,E1 3928.067,E2 3928.067} C_VEL
LIN {X 0,Y 530.188,Z 691.44,A -85,B 0,C 180,E1 3937.289,E2 3937.289} C_VEL
LIN {X 0,Y 530.575,Z 691.44,A -85,B 0,C 180,E1 3945.946,E2 3945.946} C_VEL
LIN {X 0,Y 530.889,Z 691.44,A -85,B 0,C 180,E1 3954.271,E2 3954.271} C_VEL
LIN {X 0,Y 531.015,Z 691.44,A -85,B 0,C 180,E1 3960.83,E2 3960.83} C_VEL
LIN {X 0,Y 530.753,Z 691.44,A -85,B 0,C 180,E1 3969.44,E2 3969.44} C_VEL
LIN {X 0,Y 530.658,Z 691.44,A -85,B 0,C 180,E1 3977.48,E2 3977.48} C_VEL
LIN {X 0,Y 530.654,Z 692.972,A -85,B 0,C 180,E1 3983.056,E2 3983.056} C_VEL
LIN {X 0,Y 545.154,Z 725.715,A -85,B 0,C 180,E1 3984.958,E2 3984.958} C_VEL
LIN {X 0,Y 542.299,Z 792.424,A -85,B 0,C 180,E1 3987.501,E2 3987.501} C_VEL
LIN {X 0,Y 538.541,Z 853.78,A -85,B 0,C 180,E1 3991.642,E2 3991.642} C_VEL
LIN {X 0,Y 535.008,Z 906.917,A -85,B 0,C 180,E1 3997.181,E2 3997.181} C_VEL
LIN {X 0,Y 532.874,Z 948.867,A -85,B 0,C 180,E1 4003.79,E2 4003.79} C_VEL
LIN {X 0,Y 531.734,Z 977.226,A -85,B 0,C 180,E1 4010.955,E2 4010.955} C_VEL
LIN {X 0,Y 531.072,Z 991.027,A -85,B 0,C 180,E1 4018.086,E2 4018.086} C_VEL
LIN {X 0,Y 530.985,Z 992.309,A -85,B 0,C 180,E1 4024.18,E2 4024.18} C_VEL
LIN {X 0,Y 531.041,Z 982.813,A -85,B 0,C 180,E1 4030.814,E2 4030.814} C_VEL
LIN {X 0,Y 531.649,Z 962.293,A -85,B 0,C 180,E1 4037.219,E2 4037.219} C_VEL
LIN {X 0,Y 533.463,Z 927.33,A -85,B 0,C 180,E1 4043.876,E2 4043.876} C_VEL
LIN {X 0,Y 536.701,Z 878.31,A -85,B 0,C 180,E1 4050,E2 4050} C_VEL
LIN {X 0,Y 540.858,Z 819.331,A -85,B 0,C 180,E1 4054.829,E2 4054.829} C_VEL
LIN {X 0,Y 544.392,Z 755.488,A -85,B 0,C 180,E1 4058.016,E2 4058.016} C_VEL
LIN {X 0,Y 543.808,Z 716.815,A -85,B 0,C 180,E1 4059.284,E2 4059.284} C_VEL
LIN {X 0,Y 530.841,Z 691.44,A -85,B 0,C 180,E1 4060.918,E2 4060.918} C_VEL
LIN {X 0,Y 530.608,Z 691.44,A -85,B 0,C 180,E1 4069.203,E2 4069.203} C_VEL
LIN {X 0,Y 530.454,Z 691.44,A -85,B 0,C 180,E1 4078.168,E2 4078.168} C_VEL
LIN {X 0,Y 530.398,Z 691.44,A -85,B 0,C 180,E1 4088.117,E2 4088.117} C_VEL
LIN {X 0,Y 530.521,Z 691.44,A -85,B 0,C 180,E1 4097.764,E2 4097.764} C_VEL
LIN {X 0,Y 530.462,Z 691.44,A -85,B 0,C 180,E1 4108.044,E2 4108.044} C_VEL
LIN {X 0,Y 530.538,Z 691.44,A -85,B 0,C 180,E1 4115.492,E2 4115.492} C_VEL
LIN {X 0,Y 531.464,Z 691.44,A -85,B 0,C 180,E1 4125.947,E2 4125.947} C_VEL
LIN {X 0,Y 530.978,Z 691.44,A -85,B 0,C 180,E1 4135.893,E2 4135.893} C_VEL
LIN {X 0,Y 531.205,Z 691.44,A -85,B 0,C 180,E1 4142.444,E2 4142.444} C_VEL
LIN {X 0,Y 530.809,Z 691.44,A -85,B 0,C 180,E1 4150.695,E2 4150.695} C_VEL
LIN {X 0,Y 530.573,Z 691.44,A -85,B 0,C 180,E1 4159.185,E2 4159.185} C_VEL
LIN {X 0,Y 530.404,Z 691.44,A -85,B 0,C 180,E1 4168.147,E2 4168.147} C_VEL
LIN {X 0,Y 530.211,Z 691.44,A -85,B 0,C 180,E1 4173.26,E2 4173.26} C_VEL
LIN {X 0,Y 522.147,Z 691.44,A -85,B 0,C 180,E1 4177.006,E2 4177.006} C_VEL
LIN {X 0,Y 522.477,Z 691.44,A -85,B 0,C 180,E1 4186.954,E2 4186.954} C_VEL
LIN {X 0,Y 522.479,Z 692.833,A -85,B 0,C 180,E1 4189.846,E2 4189.846} C_VEL
LIN {X 0,Y 539.323,Z 727.478,A -85,B 0,C 180,E1 4191.915,E2 4191.915} C_VEL
LIN {X 0,Y 537.413,Z 793.978,A -85,B 0,C 180,E1 4193.758,E2 4193.758} C_VEL
LIN {X 0,Y 533.379,Z 856.426,A -85,B 0,C 180,E1 4197.121,E2 4197.121} C_VEL
LIN {X 0,Y 528.796,Z 914.738,A -85,B 0,C 180,E1 4202.211,E2 4202.211} C_VEL
LIN {X 0,Y 525.352,Z 961.601,A -85,B 0,C 180,E1 4208.422,E2 4208.422} C_VEL
LIN {X 0,Y 523.564,Z 993.838,A -85,B 0,C 180,E1 4214.878,E2 4214.878} C_VEL
LIN {X 0,Y 522.95,Z 1014.286,A -85,B 0,C 180,E1 4221.657,E2 4221.657} C_VEL
LIN {X 0,Y 522.96,Z 1022.15,A -85,B 0,C 180,E1 4227.505,E2 4227.505} C_VEL
LIN {X 0,Y 523.012,Z 1020.768,A -85,B 0,C 180,E1 4234.16,E2 4234.16} C_VEL
LIN {X 0,Y 522.969,Z 1009.313,A -85,B 0,C 180,E1 4240.417,E2 4240.417} C_VEL
LIN {X 0,Y 523.924,Z 985.944,A -85,B 0,C 180,E1 4246.98,E2 4246.98} C_VEL
LIN {X 0,Y 526.316,Z 948.548,A -85,B 0,C 180,E1 4253.582,E2 4253.582} C_VEL
LIN {X 0,Y 530.239,Z 896.366,A -85,B 0,C 180,E1 4259.647,E2 4259.647} C_VEL
LIN {X 0,Y 534.84,Z 836.442,A -85,B 0,C 180,E1 4264.15,E2 4264.15} C_VEL
LIN {X 0,Y 538.499,Z 773.806,A -85,B 0,C 180,E1 4266.966,E2 4266.966} C_VEL
LIN {X 0,Y 537.912,Z 720.656,A -85,B 0,C 180,E1 4268.316,E2 4268.316} C_VEL
LIN {X 0,Y 522.605,Z 691.44,A -85,B 0,C 180,E1 4270.308,E2 4270.308} C_VEL
LIN {X 0,Y 522.182,Z 691.44,A -85,B 0,C 180,E1 4280.367,E2 4280.367} C_VEL
LIN {X 0,Y 522.301,Z 691.44,A -85,B 0,C 180,E1 4289.463,E2 4289.463} C_VEL
LIN {X 0,Y 522.212,Z 691.44,A -85,B 0,C 180,E1 4296.922,E2 4296.922} C_VEL
LIN {X 0,Y 522.593,Z 691.44,A -85,B 0,C 180,E1 4305.726,E2 4305.726} C_VEL
LIN {X 0,Y 522.907,Z 691.44,A -85,B 0,C 180,E1 4314.183,E2 4314.183} C_VEL
LIN {X 0,Y 523.021,Z 691.44,A -85,B 0,C 180,E1 4320.842,E2 4320.842} C_VEL
LIN {X 0,Y 522.763,Z 691.44,A -85,B 0,C 180,E1 4329.196,E2 4329.196} C_VEL
LIN {X 0,Y 522.662,Z 691.44,A -85,B 0,C 180,E1 4337.756,E2 4337.756} C_VEL
LIN {X 0,Y 522.824,Z 693.454,A -85,B 0,C 180,E1 4342.369,E2 4342.369} C_VEL
LIN {X 0,Y 538.659,Z 728.768,A -85,B 0,C 180,E1 4344.524,E2 4344.524} C_VEL
LIN {X 0,Y 535.366,Z 796.097,A -85,B 0,C 180,E1 4347.201,E2 4347.201} C_VEL
LIN {X 0,Y 531.085,Z 857.518,A -85,B 0,C 180,E1 4351.516,E2 4351.516} C_VEL
LIN {X 0,Y 527.238,Z 909.827,A -85,B 0,C 180,E1 4357.19,E2 4357.19} C_VEL
LIN {X 0,Y 524.989,Z 950.012,A -85,B 0,C 180,E1 4363.74,E2 4363.74} C_VEL
LIN {X 0,Y 523.665,Z 978.075,A -85,B 0,C 180,E1 4371.09,E2 4371.09} C_VEL
LIN {X 0,Y 523.199,Z 990.536,A -85,B 0,C 180,E1 4377.547,E2 4377.547} C_VEL
LIN {X 0,Y 522.997,Z 991.751,A -85,B 0,C 180,E1 4385.118,E2 4385.118} C_VEL
LIN {X 0,Y 522.967,Z 980.757,A -85,B 0,C 180,E1 4391.823,E2 4391.823} C_VEL
LIN {X 0,Y 523.682,Z 960.602,A -85,B 0,C 180,E1 4397.872,E2 4397.872} C_VEL
LIN {X 0,Y 525.751,Z 926.008,A -85,B 0,C 180,E1 4404.427,E2 4404.427} C_VEL
LIN {X 0,Y 529.438,Z 876.477,A -85,B 0,C 180,E1 4410.616,E2 4410.616} C_VEL
LIN {X 0,Y 534.089,Z 817.845,A -85,B 0,C 180,E1 4415.401,E2 4415.401} C_VEL
LIN {X 0,Y 537.881,Z 755.46,A -85,B 0,C 180,E1 4418.523,E2 4418.523} C_VEL
LIN {X 0,Y 537.502,Z 720.037,A -85,B 0,C 180,E1 4419.72,E2 4419.72} C_VEL
LIN {X 0,Y 522.782,Z 691.44,A -85,B 0,C 180,E1 4421.725,E2 4421.725} C_VEL
LIN {X 0,Y 522.607,Z 691.44,A -85,B 0,C 180,E1 4429.509,E2 4429.509} C_VEL
LIN {X 0,Y 522.477,Z 691.44,A -85,B 0,C 180,E1 4438.638,E2 4438.638} C_VEL
LIN {X 0,Y 522.355,Z 691.44,A -85,B 0,C 180,E1 4448.656,E2 4448.656} C_VEL
LIN {X 0,Y 522.515,Z 691.44,A -85,B 0,C 180,E1 4457.785,E2 4457.785} C_VEL
LIN {X 0,Y 522.464,Z 691.44,A -85,B 0,C 180,E1 4467.495,E2 4467.495} C_VEL
LIN {X 0,Y 522.209,Z 691.44,A -85,B 0,C 180,E1 4476.897,E2 4476.897} C_VEL
LIN {X 0,Y 523.407,Z 691.44,A -85,B 0,C 180,E1 4486.245,E2 4486.245} C_VEL
LIN {X 0,Y 523.005,Z 691.44,A -85,B 0,C 180,E1 4495.83,E2 4495.83} C_VEL
LIN {X 0,Y 523.214,Z 691.44,A -85,B 0,C 180,E1 4502.481,E2 4502.481} C_VEL
LIN {X 0,Y 522.776,Z 691.44,A -85,B 0,C 180,E1 4510.861,E2 4510.861} C_VEL
LIN {X 0,Y 522.554,Z 691.44,A -85,B 0,C 180,E1 4519.491,E2 4519.491} C_VEL
LIN {X 0,Y 522.428,Z 691.44,A -85,B 0,C 180,E1 4528.616,E2 4528.616} C_VEL
LIN {X 0,Y 522.147,Z 691.44,A -85,B 0,C 180,E1 4537.006,E2 4537.006} C_VEL
LIN {X 0,Y 514.249,Z 691.44,A -85,B 0,C 180,E1 4540.847,E2 4540.847} C_VEL
LIN {X 0,Y 514.651,Z 693.209,A -85,B 0,C 180,E1 4549.13,E2 4549.13} C_VEL
LIN {X 0,Y 533.023,Z 731.301,A -85,B 0,C 180,E1 4551.454,E2 4551.454} C_VEL
LIN {X 0,Y 530.685,Z 797.899,A -85,B 0,C 180,E1 4553.402,E2 4553.402} C_VEL
LIN {X 0,Y 526.214,Z 859.784,A -85,B 0,C 180,E1 4556.875,E2 4556.875} C_VEL
LIN {X 0,Y 521.213,Z 917.526,A -85,B 0,C 180,E1 4562.085,E2 4562.085} C_VEL
LIN {X 0,Y 517.405,Z 964.053,A -85,B 0,C 180,E1 4568.491,E2 4568.491} C_VEL
LIN {X 0,Y 515.538,Z 995.55,A -85,B 0,C 180,E1 4575.073,E2 4575.073} C_VEL
LIN {X 0,Y 515.008,Z 1014.286,A -85,B 0,C 180,E1 4581.527,E2 4581.527} C_VEL
LIN {X 0,Y 514.967,Z 1022.15,A -85,B 0,C 180,E1 4587.466,E2 4587.466} C_VEL
LIN {X 0,Y 515.007,Z 1020.768,A -85,B 0,C 180,E1 4594.224,E2 4594.224} C_VEL
LIN {X 0,Y 514.98,Z 1009.222,A -85,B 0,C 180,E1 4600.614,E2 4600.614} C_VEL
LIN {X 0,Y 516.017,Z 986.151,A -85,B 0,C 180,E1 4607.201,E2 4607.201} C_VEL
LIN {X 0,Y 518.584,Z 950.026,A -85,B 0,C 180,E1 4613.727,E2 4613.727} C_VEL
LIN {X 0,Y 522.743,Z 899.888,A -85,B 0,C 180,E1 4619.749,E2 4619.749} C_VEL
LIN {X 0,Y 527.74,Z 841.888,A -85,B 0,C 180,E1 4624.316,E2 4624.316} C_VEL
LIN {X 0,Y 531.736,Z 778.929,A -85,B 0,C 180,E1 4627.317,E2 4627.317} C_VEL
LIN {X 0,Y 531.575,Z 723.694,A -85,B 0,C 180,E1 4628.806,E2 4628.806} C_VEL
LIN {X 0,Y 514.484,Z 691.44,A -85,B 0,C 180,E1 4631.023,E2 4631.023} C_VEL
LIN {X 0,Y 514.138,Z 691.44,A -85,B 0,C 180,E1 4640.64,E2 4640.64} C_VEL
LIN {X 0,Y 514.253,Z 691.44,A -85,B 0,C 180,E1 4650.523,E2 4650.523} C_VEL
LIN {X 0,Y 514.024,Z 691.44,A -85,B 0,C 180,E1 4658.433,E2 4658.433} C_VEL
LIN {X 0,Y 514.439,Z 691.44,A -85,B 0,C 180,E1 4667.234,E2 4667.234} C_VEL
LIN {X 0,Y 514.833,Z 691.44,A -85,B 0,C 180,E1 4675.787,E2 4675.787} C_VEL
LIN {X 0,Y 514.816,Z 691.44,A -85,B 0,C 180,E1 4682.545,E2 4682.545} C_VEL
LIN {X 0,Y 514.843,Z 691.44,A -85,B 0,C 180,E1 4691.054,E2 4691.054} C_VEL
LIN {X 0,Y 514.725,Z 691.44,A -85,B 0,C 180,E1 4701.403,E2 4701.403} C_VEL
LIN {X 0,Y 532.241,Z 730.604,A -85,B 0,C 180,E1 4704.048,E2 4704.048} C_VEL
LIN {X 0,Y 528.526,Z 798.254,A -85,B 0,C 180,E1 4706.813,E2 4706.813} C_VEL
LIN {X 0,Y 523.932,Z 858.071,A -85,B 0,C 180,E1 4711.108,E2 4711.108} C_VEL
LIN {X 0,Y 519.683,Z 909.59,A -85,B 0,C 180,E1 4716.772,E2 4716.772} C_VEL
LIN {X 0,Y 517.097,Z 950.727,A -85,B 0,C 180,E1 4723.601,E2 4723.601} C_VEL
LIN {X 0,Y 515.804,Z 977.64,A -85,B 0,C 180,E1 4730.761,E2 4730.761} C_VEL
LIN {X 0,Y 515.243,Z 990.102,A -85,B 0,C 180,E1 4737.07,E2 4737.07} C_VEL
LIN {X 0,Y 514.915,Z 992.04,A -85,B 0,C 180,E1 4744.701,E2 4744.701} C_VEL
LIN {X 0,Y 515.024,Z 982.712,A -85,B 0,C 180,E1 4751.139,E2 4751.139} C_VEL
LIN {X 0,Y 515.758,Z 962.373,A -85,B 0,C 180,E1 4757.683,E2 4757.683} C_VEL
LIN {X 0,Y 517.937,Z 928.785,A -85,B 0,C 180,E1 4764.331,E2 4764.331} C_VEL
LIN {X 0,Y 521.836,Z 880.505,A -85,B 0,C 180,E1 4770.625,E2 4770.625} C_VEL
LIN {X 0,Y 526.851,Z 823.064,A -85,B 0,C 180,E1 4775.547,E2 4775.547} C_VEL
LIN {X 0,Y 531.25,Z 759.044,A -85,B 0,C 180,E1 4778.912,E2 4778.912} C_VEL
LIN {X 0,Y 531.023,Z 722.926,A -85,B 0,C 180,E1 4780.189,E2 4780.189} C_VEL
LIN {X 0,Y 514.775,Z 691.44,A -85,B 0,C 180,E1 4782.342,E2 4782.342} C_VEL
LIN {X 0,Y 514.717,Z 691.44,A -85,B 0,C 180,E1 4791.78,E2 4791.78} C_VEL
LIN {X 0,Y 514.488,Z 691.44,A -85,B 0,C 180,E1 4801.078,E2 4801.078} C_VEL
LIN {X 0,Y 514.325,Z 691.44,A -85,B 0,C 180,E1 4811.598,E2 4811.598} C_VEL
LIN {X 0,Y 514.148,Z 691.44,A -85,B 0,C 180,E1 4820.611,E2 4820.611} C_VEL
LIN {X 0,Y 514.289,Z 691.44,A -85,B 0,C 180,E1 4830.518,E2 4830.518} C_VEL
LIN {X 0,Y 514.033,Z 691.44,A -85,B 0,C 180,E1 4838.433,E2 4838.433} C_VEL
LIN {X 0,Y 515.216,Z 691.44,A -85,B 0,C 180,E1 4847.23,E2 4847.23} C_VEL
LIN {X 0,Y 515.008,Z 691.44,A -85,B 0,C 180,E1 4855.765,E2 4855.765} C_VEL
LIN {X 0,Y 515.195,Z 691.44,A -85,B 0,C 180,E1 4862.52,E2 4862.52} C_VEL
LIN {X 0,Y 514.764,Z 691.44,A -85,B 0,C 180,E1 4871.032,E2 4871.032} C_VEL
LIN {X 0,Y 514.54,Z 691.44,A -85,B 0,C 180,E1 4879.807,E2 4879.807} C_VEL
LIN {X 0,Y 514.39,Z 691.44,A -85,B 0,C 180,E1 4889.502,E2 4889.502} C_VEL
LIN {X 0,Y 514.295,Z 691.44,A -85,B 0,C 180,E1 4899.346,E2 4899.346} C_VEL
LIN {X 0,Y 514.249,Z 691.44,A -85,B 0,C 180,E1 4900.847,E2 4900.847} C_VEL
LIN {X 0,Y 506.186,Z 691.44,A -85,B 0,C 180,E1 4904.725,E2 4904.725} C_VEL
LIN {X 0,Y 506.559,Z 692.701,A -85,B 0,C 180,E1 4908.342,E2 4908.342} C_VEL
LIN {X 0,Y 526.76,Z 732.859,A -85,B 0,C 180,E1 4910.941,E2 4910.941} C_VEL
LIN {X 0,Y 524.168,Z 798.677,A -85,B 0,C 180,E1 4912.907,E2 4912.907} C_VEL
LIN {X 0,Y 519.201,Z 861.206,A -85,B 0,C 180,E1 4916.485,E2 4916.485} C_VEL
LIN {X 0,Y 513.815,Z 918.211,A -85,B 0,C 180,E1 4921.729,E2 4921.729} C_VEL
LIN {X 0,Y 509.745,Z 964.051,A -85,B 0,C 180,E1 4928.152,E2 4928.152} C_VEL
LIN {X 0,Y 507.656,Z 995.551,A -85,B 0,C 180,E1 4934.836,E2 4934.836} C_VEL
LIN {X 0,Y 507.064,Z 1014.286,A -85,B 0,C 180,E1 4941.393,E2 4941.393} C_VEL
LIN {X 0,Y 506.98,Z 1022.15,A -85,B 0,C 180,E1 4947.426,E2 4947.426} C_VEL
LIN {X 0,Y 507.017,Z 1020.768,A -85,B 0,C 180,E1 4954.291,E2 4954.291} C_VEL
LIN {X 0,Y 507.018,Z 1009.224,A -85,B 0,C 180,E1 4960.782,E2 4960.782} C_VEL
LIN {X 0,Y 508.117,Z 986.15,A -85,B 0,C 180,E1 4967.477,E2 4967.477} C_VEL
LIN {X 0,Y 510.93,Z 950.311,A -85,B 0,C 180,E1 4974.06,E2 4974.06} C_VEL
LIN {X 0,Y 515.398,Z 901.467,A -85,B 0,C 180,E1 4980.05,E2 4980.05} C_VEL
LIN {X 0,Y 520.87,Z 843.474,A -85,B 0,C 180,E1 4984.727,E2 4984.727} C_VEL
LIN {X 0,Y 525.29,Z 779.859,A -85,B 0,C 180,E1 4987.817,E2 4987.817} C_VEL
LIN {X 0,Y 525.515,Z 726.844,A -85,B 0,C 180,E1 4989.285,E2 4989.285} C_VEL
LIN {X 0,Y 506.374,Z 691.44,A -85,B 0,C 180,E1 4991.774,E2 4991.774} C_VEL
LIN {X 0,Y 506.21,Z 691.44,A -85,B 0,C 180,E1 4999.9,E2 4999.9} C_VEL
LIN {X 0,Y 506.295,Z 691.44,A -85,B 0,C 180,E1 5008.679,E2 5008.679} C_VEL
LIN {X 0,Y 506.031,Z 691.44,A -85,B 0,C 180,E1 5018.004,E2 5018.004} C_VEL
LIN {X 0,Y 506.433,Z 691.44,A -85,B 0,C 180,E1 5027.029,E2 5027.029} C_VEL
LIN {X 0,Y 506.835,Z 691.44,A -85,B 0,C 180,E1 5035.72,E2 5035.72} C_VEL
LIN {X 0,Y 506.818,Z 691.44,A -85,B 0,C 180,E1 5042.585,E2 5042.585} C_VEL
LIN {X 0,Y 506.838,Z 691.44,A -85,B 0,C 180,E1 5051.231,E2 5051.231} C_VEL
LIN {X 0,Y 506.976,Z 693.242,A -85,B 0,C 180,E1 5060.884,E2 5060.884} C_VEL
LIN {X 0,Y 525.826,Z 734.556,A -85,B 0,C 180,E1 5063.623,E2 5063.623} C_VEL
LIN {X 0,Y 521.536,Z 802.08,A -85,B 0,C 180,E1 5066.52,E2 5066.52} C_VEL
LIN {X 0,Y 516.387,Z 862.586,A -85,B 0,C 180,E1 5071.053,E2 5071.053} C_VEL
LIN {X 0,Y 511.86,Z 913.215,A -85,B 0,C 180,E1 5076.878,E2 5076.878} C_VEL
LIN {X 0,Y 509.085,Z 953.36,A -85,B 0,C 180,E1 5083.871,E2 5083.871} C_VEL
LIN {X 0,Y 507.513,Z 979.813,A -85,B 0,C 180,E1 5091.393,E2 5091.393} C_VEL
LIN {X 0,Y 506.919,Z 991.627,A -85,B 0,C 180,E1 5098.552,E2 5098.552} C_VEL
LIN {X 0,Y 507.032,Z 990.874,A -85,B 0,C 180,E1 5106.168,E2 5106.168} C_VEL
LIN {X 0,Y 507.313,Z 977.221,A -85,B 0,C 180,E1 5113.49,E2 5113.49} C_VEL
LIN {X 0,Y 508.845,Z 949.976,A -85,B 0,C 180,E1 5120.776,E2 5120.776} C_VEL
LIN {X 0,Y 512.156,Z 908.674,A -85,B 0,C 180,E1 5127.665,E2 5127.665} C_VEL
LIN {X 0,Y 517.038,Z 855.144,A -85,B 0,C 180,E1 5133.545,E2 5133.545} C_VEL
LIN {X 0,Y 522.306,Z 793.617,A -85,B 0,C 180,E1 5137.856,E2 5137.856} C_VEL
LIN {X 0,Y 524.711,Z 726.275,A -85,B 0,C 180,E1 5140.635,E2 5140.635} C_VEL
LIN {X 0,Y 506.786,Z 691.44,A -85,B 0,C 180,E1 5143.324,E2 5143.324} C_VEL
LIN {X 0,Y 506.714,Z 691.44,A -85,B 0,C 180,E1 5151.986,E2 5151.986} C_VEL
LIN {X 0,Y 506.397,Z 691.44,A -85,B 0,C 180,E1 5161.631,E2 5161.631} C_VEL
LIN {X 0,Y 506.303,Z 691.44,A -85,B 0,C 180,E1 5170.158,E2 5170.158} C_VEL
LIN {X 0,Y 506.196,Z 691.44,A -85,B 0,C 180,E1 5179.868,E2 5179.868} C_VEL
LIN {X 0,Y 506.335,Z 691.44,A -85,B 0,C 180,E1 5188.673,E2 5188.673} C_VEL
LIN {X 0,Y 506.041,Z 691.44,A -85,B 0,C 180,E1 5197.979,E2 5197.979} C_VEL
LIN {X 0,Y 507.207,Z 691.44,A -85,B 0,C 180,E1 5207.025,E2 5207.025} C_VEL
LIN {X 0,Y 507.009,Z 691.44,A -85,B 0,C 180,E1 5215.698,E2 5215.698} C_VEL
LIN {X 0,Y 507.194,Z 691.44,A -85,B 0,C 180,E1 5222.56,E2 5222.56} C_VEL
LIN {X 0,Y 506.738,Z 691.44,A -85,B 0,C 180,E1 5231.209,E2 5231.209} C_VEL
LIN {X 0,Y 506.552,Z 691.44,A -85,B 0,C 180,E1 5240.133,E2 5240.133} C_VEL
LIN {X 0,Y 506.401,Z 691.44,A -85,B 0,C 180,E1 5249.61,E2 5249.61} C_VEL
LIN {X 0,Y 506.24,Z 691.44,A -85,B 0,C 180,E1 5260.143,E2 5260.143} C_VEL
LIN {X 0,Y 506.186,Z 691.44,A -85,B 0,C 180,E1 5264.725,E2 5264.725} C_VEL
LIN {X 0,Y 498.321,Z 691.44,A -85,B 0,C 180,E1 5267.31,E2 5267.31} C_VEL
LIN {X 0,Y 520.527,Z 736.172,A -85,B 0,C 180,E1 5270.451,E2 5270.451} C_VEL
LIN {X 0,Y 517.609,Z 800.676,A -85,B 0,C 180,E1 5272.451,E2 5272.451} C_VEL
LIN {X 0,Y 512.158,Z 863.279,A -85,B 0,C 180,E1 5276.134,E2 5276.134} C_VEL
LIN {X 0,Y 506.45,Z 918.772,A -85,B 0,C 180,E1 5281.351,E2 5281.351} C_VEL
LIN {X 0,Y 501.926,Z 965.378,A -85,B 0,C 180,E1 5288.027,E2 5288.027} C_VEL
LIN {X 0,Y 499.813,Z 995.552,A -85,B 0,C 180,E1 5294.592,E2 5294.592} C_VEL
LIN {X 0,Y 499.04,Z 1014.791,A -85,B 0,C 180,E1 5301.521,E2 5301.521} C_VEL
LIN {X 0,Y 498.987,Z 1022.15,A -85,B 0,C 180,E1 5307.385,E2 5307.385} C_VEL
LIN {X 0,Y 499.014,Z 1020.768,A -85,B 0,C 180,E1 5314.36,E2 5314.36} C_VEL
LIN {X 0,Y 499.086,Z 1008.073,A -85,B 0,C 180,E1 5321.399,E2 5321.399} C_VEL
LIN {X 0,Y 500.423,Z 984.272,A -85,B 0,C 180,E1 5328.192,E2 5328.192} C_VEL
LIN {X 0,Y 503.586,Z 946.835,A -85,B 0,C 180,E1 5334.974,E2 5334.974} C_VEL
LIN {X 0,Y 508.902,Z 895.488,A -85,B 0,C 180,E1 5341.118,E2 5341.118} C_VEL
LIN {X 0,Y 514.8,Z 835.492,A -85,B 0,C 180,E1 5345.741,E2 5345.741} C_VEL
LIN {X 0,Y 519.39,Z 773.464,A -85,B 0,C 180,E1 5348.583,E2 5348.583} C_VEL
LIN {X 0,Y 519.195,Z 729.766,A -85,B 0,C 180,E1 5349.802,E2 5349.802} C_VEL
LIN {X 0,Y 498.252,Z 691.44,A -85,B 0,C 180,E1 5352.565,E2 5352.565} C_VEL
LIN {X 0,Y 498.024,Z 691.44,A -85,B 0,C 180,E1 5361.373,E2 5361.373} C_VEL
LIN {X 0,Y 498.256,Z 691.44,A -85,B 0,C 180,E1 5370.232,E2 5370.232} C_VEL
LIN {X 0,Y 498.012,Z 691.44,A -85,B 0,C 180,E1 5379.506,E2 5379.506} C_VEL
LIN {X 0,Y 498.474,Z 691.44,A -85,B 0,C 180,E1 5386.818,E2 5386.818} C_VEL
LIN {X 0,Y 498.83,Z 691.44,A -85,B 0,C 180,E1 5395.651,E2 5395.651} C_VEL
LIN {X 0,Y 498.819,Z 691.44,A -85,B 0,C 180,E1 5402.627,E2 5402.627} C_VEL
LIN {X 0,Y 498.829,Z 691.44,A -85,B 0,C 180,E1 5411.413,E2 5411.413} C_VEL
LIN {X 0,Y 498.924,Z 693.02,A -85,B 0,C 180,E1 5420.08,E2 5420.08} C_VEL
LIN {X 0,Y 519.427,Z 737.407,A -85,B 0,C 180,E1 5423.164,E2 5423.164} C_VEL
LIN {X 0,Y 514.83,Z 803.012,A -85,B 0,C 180,E1 5426.049,E2 5426.049} C_VEL
LIN {X 0,Y 509.231,Z 863.039,A -85,B 0,C 180,E1 5430.615,E2 5430.615} C_VEL
LIN {X 0,Y 504.226,Z 914.307,A -85,B 0,C 180,E1 5436.632,E2 5436.632} C_VEL
LIN {X 0,Y 501.1,Z 954.708,A -85,B 0,C 180,E1 5443.883,E2 5443.883} C_VEL
LIN {X 0,Y 499.473,Z 980.418,A -85,B 0,C 180,E1 5451.475,E2 5451.475} C_VEL
LIN {X 0,Y 499.031,Z 991.046,A -85,B 0,C 180,E1 5457.847,E2 5457.847} C_VEL
LIN {X 0,Y 498.794,Z 992.577,A -85,B 0,C 180,E1 5463.822,E2 5463.822} C_VEL
LIN {X 0,Y 499.112,Z 984.135,A -85,B 0,C 180,E1 5470.762,E2 5470.762} C_VEL
LIN {X 0,Y 499.873,Z 964.156,A -85,B 0,C 180,E1 5477.731,E2 5477.731} C_VEL
LIN {X 0,Y 502.448,Z 929.788,A -85,B 0,C 180,E1 5484.889,E2 5484.889} C_VEL
LIN {X 0,Y 507.089,Z 882.672,A -85,B 0,C 180,E1 5491.287,E2 5491.287} C_VEL
LIN {X 0,Y 512.958,Z 825.757,A -85,B 0,C 180,E1 5496.37,E2 5496.37} C_VEL
LIN {X 0,Y 518.13,Z 762.789,A -85,B 0,C 180,E1 5499.835,E2 5499.835} C_VEL
LIN {X 0,Y 518.398,Z 729.67,A -85,B 0,C 180,E1 5501.091,E2 5501.091} C_VEL
LIN {X 0,Y 498.83,Z 691.44,A -85,B 0,C 180,E1 5504.087,E2 5504.087} C_VEL
LIN {X 0,Y 498.599,Z 691.44,A -85,B 0,C 180,E1 5514.262,E2 5514.262} C_VEL
LIN {X 0,Y 498.163,Z 691.44,A -85,B 0,C 180,E1 5524.304,E2 5524.304} C_VEL
LIN {X 0,Y 498.157,Z 691.44,A -85,B 0,C 180,E1 5534.286,E2 5534.286} C_VEL
LIN {X 0,Y 498.133,Z 691.44,A -85,B 0,C 180,E1 5543.837,E2 5543.837} C_VEL
LIN {X 0,Y 498.459,Z 691.44,A -85,B 0,C 180,E1 5553.916,E2 5553.916} C_VEL
LIN {X 0,Y 499.212,Z 691.44,A -85,B 0,C 180,E1 5565.018,E2 5565.018} C_VEL
LIN {X 0,Y 499.008,Z 691.44,A -85,B 0,C 180,E1 5575.629,E2 5575.629} C_VEL
LIN {X 0,Y 499.175,Z 691.44,A -85,B 0,C 180,E1 5582.601,E2 5582.601} C_VEL
LIN {X 0,Y 498.714,Z 691.44,A -85,B 0,C 180,E1 5591.392,E2 5591.392} C_VEL
LIN {X 0,Y 498.536,Z 691.44,A -85,B 0,C 180,E1 5600.471,E2 5600.471} C_VEL
LIN {X 0,Y 498.381,Z 691.44,A -85,B 0,C 180,E1 5610.135,E2 5610.135} C_VEL
LIN {X 0,Y 498.15,Z 691.44,A -85,B 0,C 180,E1 5620.885,E2 5620.885} C_VEL
LIN {X 0,Y 498.321,Z 691.44,A -85,B 0,C 180,E1 5627.31,E2 5627.31} C_VEL
LIN {X 0,Y 503.086,Z 701.503,A -85,B 0,C 180,E1 5628.162,E2 5628.162} C_VEL
LIN {X 0,Y 506.932,Z 722.853,A -85,B 0,C 180,E1 5628.934,E2 5628.934} C_VEL
LIN {X 0,Y 514.289,Z 739.453,A -85,B 0,C 180,E1 5629.957,E2 5629.957} C_VEL
LIN {X 0,Y 510.967,Z 803.658,A -85,B 0,C 180,E1 5632.029,E2 5632.029} C_VEL
LIN {X 0,Y 505.016,Z 866.581,A -85,B 0,C 180,E1 5635.869,E2 5635.869} C_VEL
LIN {X 0,Y 498.701,Z 922.61,A -85,B 0,C 180,E1 5641.361,E2 5641.361} C_VEL
LIN {X 0,Y 494.113,Z 966.672,A -85,B 0,C 180,E1 5647.899,E2 5647.899} C_VEL
LIN {X 0,Y 491.735,Z 997.105,A -85,B 0,C 180,E1 5654.791,E2 5654.791} C_VEL
LIN {X 0,Y 491.069,Z 1014.827,A -85,B 0,C 180,E1 5661.402,E2 5661.402} C_VEL
LIN {X 0,Y 491.003,Z 1022.149,A -85,B 0,C 180,E1 5667.342,E2 5667.342} C_VEL
LIN {X 0,Y 491.031,Z 1020.768,A -85,B 0,C 180,E1 5674.431,E2 5674.431} C_VEL
LIN {X 0,Y 491.142,Z 1008.074,A -85,B 0,C 180,E1 5681.586,E2 5681.586} C_VEL
LIN {X 0,Y 492.618,Z 984.112,A -85,B 0,C 180,E1 5688.528,E2 5688.528} C_VEL
LIN {X 0,Y 496.141,Z 946.181,A -85,B 0,C 180,E1 5695.473,E2 5695.473} C_VEL
LIN {X 0,Y 501.883,Z 894.633,A -85,B 0,C 180,E1 5701.693,E2 5701.693} C_VEL
LIN {X 0,Y 508.268,Z 834.593,A -85,B 0,C 180,E1 5706.335,E2 5706.335} C_VEL
LIN {X 0,Y 513.132,Z 772.423,A -85,B 0,C 180,E1 5709.173,E2 5709.173} C_VEL
LIN {X 0,Y 512.874,Z 732.745,A -85,B 0,C 180,E1 5710.308,E2 5710.308} C_VEL
LIN {X 0,Y 490.189,Z 691.44,A -85,B 0,C 180,E1 5713.359,E2 5713.359} C_VEL
LIN {X 0,Y 489.984,Z 691.44,A -85,B 0,C 180,E1 5722.877,E2 5722.877} C_VEL
LIN {X 0,Y 490.318,Z 691.44,A -85,B 0,C 180,E1 5731.897,E2 5731.897} C_VEL
LIN {X 0,Y 490.56,Z 691.44,A -85,B 0,C 180,E1 5742.928,E2 5742.928} C_VEL
LIN {X 0,Y 491.038,Z 691.44,A -85,B 0,C 180,E1 5752.021,E2 5752.021} C_VEL
LIN {X 0,Y 491.025,Z 691.44,A -85,B 0,C 180,E1 5760.897,E2 5760.897} C_VEL
LIN {X 0,Y 490.743,Z 691.44,A -85,B 0,C 180,E1 5769.801,E2 5769.801} C_VEL
LIN {X 0,Y 490.782,Z 692.715,A -85,B 0,C 180,E1 5779.228,E2 5779.228} C_VEL
LIN {X 0,Y 513.021,Z 739.909,A -85,B 0,C 180,E1 5782.678,E2 5782.678} C_VEL
LIN {X 0,Y 507.985,Z 805.747,A -85,B 0,C 180,E1 5785.673,E2 5785.673} C_VEL
LIN {X 0,Y 501.82,Z 866.661,A -85,B 0,C 180,E1 5790.471,E2 5790.471} C_VEL
LIN {X 0,Y 496.477,Z 916.788,A -85,B 0,C 180,E1 5796.588,E2 5796.588} C_VEL
LIN {X 0,Y 493.173,Z 955.692,A -85,B 0,C 180,E1 5803.815,E2 5803.815} C_VEL
LIN {X 0,Y 491.526,Z 980.63,A -85,B 0,C 180,E1 5811.397,E2 5811.397} C_VEL
LIN {X 0,Y 490.932,Z 991.422,A -85,B 0,C 180,E1 5818.211,E2 5818.211} C_VEL
LIN {X 0,Y 490.991,Z 991.384,A -85,B 0,C 180,E1 5825.74,E2 5825.74} C_VEL
LIN {X 0,Y 491.172,Z 979.665,A -85,B 0,C 180,E1 5832.931,E2 5832.931} C_VEL
LIN {X 0,Y 492.657,Z 955.141,A -85,B 0,C 180,E1 5840.246,E2 5840.246} C_VEL
LIN {X 0,Y 496.271,Z 916.553,A -85,B 0,C 180,E1 5847.371,E2 5847.371} C_VEL
LIN {X 0,Y 501.947,Z 864.097,A -85,B 0,C 180,E1 5853.693,E2 5853.693} C_VEL
LIN {X 0,Y 508.348,Z 803.346,A -85,B 0,C 180,E1 5858.369,E2 5858.369} C_VEL
LIN {X 0,Y 513.263,Z 740.201,A -85,B 0,C 180,E1 5861.2,E2 5861.2} C_VEL
LIN {X 0,Y 506.565,Z 721.984,A -85,B 0,C 180,E1 5862.422,E2 5862.422} C_VEL
LIN {X 0,Y 490.874,Z 691.44,A -85,B 0,C 180,E1 5864.746,E2 5864.746} C_VEL
LIN {X 0,Y 490.542,Z 691.44,A -85,B 0,C 180,E1 5874.687,E2 5874.687} C_VEL
LIN {X 0,Y 490.094,Z 691.44,A -85,B 0,C 180,E1 5884.95,E2 5884.95} C_VEL
LIN {X 0,Y 490.15,Z 691.44,A -85,B 0,C 180,E1 5894.159,E2 5894.159} C_VEL
LIN {X 0,Y 489.998,Z 691.44,A -85,B 0,C 180,E1 5902.848,E2 5902.848} C_VEL
LIN {X 0,Y 490.364,Z 691.44,A -85,B 0,C 180,E1 5911.888,E2 5911.888} C_VEL
LIN {X 0,Y 490.743,Z 691.44,A -85,B 0,C 180,E1 5922.909,E2 5922.909} C_VEL
LIN {X 0,Y 490.909,Z 691.44,A -85,B 0,C 180,E1 5931.994,E2 5931.994} C_VEL
LIN {X 0,Y 491.175,Z 691.44,A -85,B 0,C 180,E1 5942.643,E2 5942.643} C_VEL
LIN {X 0,Y 490.694,Z 691.44,A -85,B 0,C 180,E1 5951.581,E2 5951.581} C_VEL
LIN {X 0,Y 490.542,Z 691.44,A -85,B 0,C 180,E1 5960.82,E2 5960.82} C_VEL
LIN {X 0,Y 490.275,Z 691.44,A -85,B 0,C 180,E1 5970.687,E2 5970.687} C_VEL
LIN {X 0,Y 490.125,Z 691.44,A -85,B 0,C 180,E1 5980.658,E2 5980.658} C_VEL
LIN {X 0,Y 490.393,Z 692.867,A -85,B 0,C 180,E1 5986.685,E2 5986.685} C_VEL
LIN {X 0,Y 506.932,Z 722.853,A -85,B 0,C 180,E1 5988.934,E2 5988.934} C_VEL
LIN {X 0,Y 509.183,Z 739.643,A -85,B 0,C 180,E1 5989.489,E2 5989.489} C_VEL
LIN {X 0,Y 507.415,Z 757.96,A -85,B 0,C 180,E1 5989.817,E2 5989.817} C_VEL
LIN {X 0,Y 502.907,Z 822.185,A -85,B 0,C 180,E1 5992.401,E2 5992.401} C_VEL
LIN {X 0,Y 496.381,Z 882.922,A -85,B 0,C 180,E1 5996.711,E2 5996.711} C_VEL
LIN {X 0,Y 489.644,Z 937.928,A -85,B 0,C 180,E1 6002.902,E2 6002.902} C_VEL
LIN {X 0,Y 485.361,Z 979.523,A -85,B 0,C 180,E1 6010.137,E2 6010.137} C_VEL
LIN {X 0,Y 483.639,Z 1006.915,A -85,B 0,C 180,E1 6017.771,E2 6017.771} C_VEL
LIN {X 0,Y 483.467,Z 1020.766,A -85,B 0,C 180,E1 6025.499,E2 6025.499} C_VEL
LIN {X 0,Y 483.253,Z 1022.15,A -85,B 0,C 180,E1 6032.7,E2 6032.7} C_VEL
LIN {X 0,Y 483.13,Z 1012.357,A -85,B 0,C 180,E1 6039.948,E2 6039.948} C_VEL
LIN {X 0,Y 484.351,Z 990.342,A -85,B 0,C 180,E1 6047.317,E2 6047.317} C_VEL
LIN {X 0,Y 487.696,Z 955.602,A -85,B 0,C 180,E1 6054.397,E2 6054.397} C_VEL
LIN {X 0,Y 493.462,Z 906.191,A -85,B 0,C 180,E1 6061.006,E2 6061.006} C_VEL
LIN {X 0,Y 500.438,Z 847.387,A -85,B 0,C 180,E1 6066.062,E2 6066.062} C_VEL
LIN {X 0,Y 505.871,Z 785.523,A -85,B 0,C 180,E1 6069.276,E2 6069.276} C_VEL
LIN {X 0,Y 506.735,Z 736.125,A -85,B 0,C 180,E1 6070.805,E2 6070.805} C_VEL
LIN {X 0,Y 482.173,Z 691.44,A -85,B 0,C 180,E1 6074.314,E2 6074.314} C_VEL
LIN {X 0,Y 482.039,Z 691.44,A -85,B 0,C 180,E1 6084.408,E2 6084.408} C_VEL
LIN {X 0,Y 482.259,Z 691.44,A -85,B 0,C 180,E1 6094.884,E2 6094.884} C_VEL
LIN {X 0,Y 482.565,Z 691.44,A -85,B 0,C 180,E1 6104.514,E2 6104.514} C_VEL
LIN {X 0,Y 482.912,Z 691.44,A -85,B 0,C 180,E1 6113.7,E2 6113.7} C_VEL
LIN {X 0,Y 483.019,Z 691.44,A -85,B 0,C 180,E1 6120.912,E2 6120.912} C_VEL
LIN {X 0,Y 482.748,Z 691.44,A -85,B 0,C 180,E1 6129.965,E2 6129.965} C_VEL
LIN {X 0,Y 482.652,Z 692.323,A -85,B 0,C 180,E1 6138.332,E2 6138.332} C_VEL
LIN {X 0,Y 506.69,Z 742.971,A -85,B 0,C 180,E1 6142.204,E2 6142.204} C_VEL
LIN {X 0,Y 501.19,Z 808.359,A -85,B 0,C 180,E1 6145.28,E2 6145.28} C_VEL
LIN {X 0,Y 494.604,Z 867.897,A -85,B 0,C 180,E1 6150.097,E2 6150.097} C_VEL
LIN {X 0,Y 488.829,Z 917.883,A -85,B 0,C 180,E1 6156.341,E2 6156.341} C_VEL
LIN {X 0,Y 485.158,Z 957.262,A -85,B 0,C 180,E1 6163.89,E2 6163.89} C_VEL
LIN {X 0,Y 483.39,Z 981.806,A -85,B 0,C 180,E1 6171.739,E2 6171.739} C_VEL
LIN {X 0,Y 482.826,Z 991.897,A -85,B 0,C 180,E1 6178.761,E2 6178.761} C_VEL
LIN {X 0,Y 483.128,Z 990.403,A -85,B 0,C 180,E1 6186.881,E2 6186.881} C_VEL
LIN {X 0,Y 484.054,Z 974.612,A -85,B 0,C 180,E1 6195.01,E2 6195.01} C_VEL
LIN {X 0,Y 486.25,Z 943.577,A -85,B 0,C 180,E1 6203.054,E2 6203.054} C_VEL
LIN {X 0,Y 490.768,Z 900.786,A -85,B 0,C 180,E1 6210,E2 6210} C_VEL
LIN {X 0,Y 497.066,Z 846.543,A -85,B 0,C 180,E1 6215.805,E2 6215.805} C_VEL
LIN {X 0,Y 503.465,Z 783.671,A -85,B 0,C 180,E1 6220.036,E2 6220.036} C_VEL
LIN {X 0,Y 505.781,Z 736.292,A -85,B 0,C 180,E1 6222.038,E2 6222.038} C_VEL
LIN {X 0,Y 482.805,Z 691.44,A -85,B 0,C 180,E1 6225.755,E2 6225.755} C_VEL
LIN {X 0,Y 482.451,Z 691.44,A -85,B 0,C 180,E1 6235.129,E2 6235.129} C_VEL
LIN {X 0,Y 482.133,Z 691.44,A -85,B 0,C 180,E1 6243.483,E2 6243.483} C_VEL
LIN {X 0,Y 482.141,Z 691.44,A -85,B 0,C 180,E1 6252.59,E2 6252.59} C_VEL
LIN {X 0,Y 481.996,Z 691.44,A -85,B 0,C 180,E1 6262.123,E2 6262.123} C_VEL
LIN {X 0,Y 482.214,Z 691.44,A -85,B 0,C 180,E1 6270.801,E2 6270.801} C_VEL
LIN {X 0,Y 482.192,Z 691.44,A -85,B 0,C 180,E1 6280.697,E2 6280.697} C_VEL
LIN {X 0,Y 482.956,Z 691.44,A -85,B 0,C 180,E1 6288.206,E2 6288.206} C_VEL
LIN {X 0,Y 482.82,Z 691.44,A -85,B 0,C 180,E1 6297.286,E2 6297.286} C_VEL
LIN {X 0,Y 482.807,Z 691.44,A -85,B 0,C 180,E1 6304.493,E2 6304.493} C_VEL
LIN {X 0,Y 482.732,Z 691.44,A -85,B 0,C 180,E1 6313.62,E2 6313.62} C_VEL
LIN {X 0,Y 482.545,Z 691.44,A -85,B 0,C 180,E1 6323.127,E2 6323.127} C_VEL
LIN {X 0,Y 482.059,Z 691.44,A -85,B 0,C 180,E1 6333.461,E2 6333.461} C_VEL
LIN {X 0,Y 482.074,Z 691.44,A -85,B 0,C 180,E1 6342.561,E2 6342.561} C_VEL
LIN {X 0,Y 482.433,Z 693.326,A -85,B 0,C 180,E1 6345.819,E2 6345.819} C_VEL
LIN {X 0,Y 508.06,Z 741.896,A -85,B 0,C 180,E1 6349.432,E2 6349.432} C_VEL
LIN {X 0,Y 507.415,Z 757.96,A -85,B 0,C 180,E1 6349.817,E2 6349.817} C_VEL
LIN {X 0,Y 498.929,Z 791.931,A -85,B 0,C 180,E1 6350.391,E2 6350.391} C_VEL
LIN {X 0,Y 492.562,Z 856.875,A -85,B 0,C 180,E1 6354.034,E2 6354.034} C_VEL
LIN {X 0,Y 485.304,Z 914.919,A -85,B 0,C 180,E1 6359.493,E2 6359.493} C_VEL
LIN {X 0,Y 479.569,Z 961.994,A -85,B 0,C 180,E1 6366.318,E2 6366.318} C_VEL
LIN {X 0,Y 476.283,Z 995.554,A -85,B 0,C 180,E1 6373.811,E2 6373.811} C_VEL
LIN {X 0,Y 475.243,Z 1014.285,A -85,B 0,C 180,E1 6380.812,E2 6380.812} C_VEL
LIN {X 0,Y 475.026,Z 1022.149,A -85,B 0,C 180,E1 6387.253,E2 6387.253} C_VEL
LIN {X 0,Y 475.03,Z 1020.768,A -85,B 0,C 180,E1 6394.581,E2 6394.581} C_VEL
LIN {X 0,Y 475.271,Z 1008.073,A -85,B 0,C 180,E1 6401.979,E2 6401.979} C_VEL
LIN {X 0,Y 477.262,Z 982.655,A -85,B 0,C 180,E1 6409.504,E2 6409.504} C_VEL
LIN {X 0,Y 481.882,Z 941.663,A -85,B 0,C 180,E1 6416.994,E2 6416.994} C_VEL
LIN {X 0,Y 488.517,Z 889.65,A -85,B 0,C 180,E1 6423.189,E2 6423.189} C_VEL
LIN {X 0,Y 495.497,Z 831.069,A -85,B 0,C 180,E1 6427.648,E2 6427.648} C_VEL
LIN {X 0,Y 500.86,Z 767.508,A -85,B 0,C 180,E1 6430.445,E2 6430.445} C_VEL
LIN {X 0,Y 500.268,Z 738.727,A -85,B 0,C 180,E1 6431.366,E2 6431.366} C_VEL
LIN {X 0,Y 474.146,Z 691.44,A -85,B 0,C 180,E1 6435.139,E2 6435.139} C_VEL
LIN {X 0,Y 474.064,Z 691.44,A -85,B 0,C 180,E1 6445.958,E2 6445.958} C_VEL
LIN {X 0,Y 474.106,Z 691.44,A -85,B 0,C 180,E1 6455.82,E2 6455.82} C_VEL
LIN {X 0,Y 474.454,Z 691.44,A -85,B 0,C 180,E1 6466.138,E2 6466.138} C_VEL
LIN {X 0,Y 474.839,Z 691.44,A -85,B 0,C 180,E1 6475.431,E2 6475.431} C_VEL
LIN {X 0,Y 474.824,Z 691.44,A -85,B 0,C 180,E1 6482.759,E2 6482.759} C_VEL
LIN {X 0,Y 474.817,Z 691.44,A -85,B 0,C 180,E1 6491.999,E2 6491.999} C_VEL
LIN {X 0,Y 474.773,Z 693.108,A -85,B 0,C 180,E1 6497.443,E2 6497.443} C_VEL
LIN {X 0,Y 500.427,Z 745.276,A -85,B 0,C 180,E1 6501.693,E2 6501.693} C_VEL
LIN {X 0,Y 494.329,Z 811.7,A -85,B 0,C 180,E1 6504.927,E2 6504.927} C_VEL
LIN {X 0,Y 487.149,Z 871.061,A -85,B 0,C 180,E1 6509.915,E2 6509.915} C_VEL
LIN {X 0,Y 481.043,Z 920.43,A -85,B 0,C 180,E1 6516.317,E2 6516.317} C_VEL
LIN {X 0,Y 477.185,Z 958.515,A -85,B 0,C 180,E1 6523.89,E2 6523.89} C_VEL
LIN {X 0,Y 475.312,Z 982.783,A -85,B 0,C 180,E1 6532.022,E2 6532.022} C_VEL
LIN {X 0,Y 474.836,Z 991.495,A -85,B 0,C 180,E1 6538.174,E2 6538.174} C_VEL
LIN {X 0,Y 475.013,Z 990.874,A -85,B 0,C 180,E1 6546.463,E2 6546.463} C_VEL
LIN {X 0,Y 475.708,Z 977.218,A -85,B 0,C 180,E1 6554.267,E2 6554.267} C_VEL
LIN {X 0,Y 478.17,Z 948.013,A -85,B 0,C 180,E1 6562.478,E2 6562.478} C_VEL
LIN {X 0,Y 482.78,Z 905.886,A -85,B 0,C 180,E1 6569.775,E2 6569.775} C_VEL
LIN {X 0,Y 489.436,Z 852.325,A -85,B 0,C 180,E1 6575.831,E2 6575.831} C_VEL
LIN {X 0,Y 496.484,Z 790.734,A -85,B 0,C 180,E1 6580.234,E2 6580.234} C_VEL
LIN {X 0,Y 499.383,Z 739.271,A -85,B 0,C 180,E1 6582.547,E2 6582.547} C_VEL
LIN {X 0,Y 474.754,Z 691.44,A -85,B 0,C 180,E1 6586.707,E2 6586.707} C_VEL
LIN {X 0,Y 474.39,Z 691.44,A -85,B 0,C 180,E1 6595.587,E2 6595.587} C_VEL
LIN {X 0,Y 473.987,Z 691.44,A -85,B 0,C 180,E1 6605.277,E2 6605.277} C_VEL
LIN {X 0,Y 474.051,Z 691.44,A -85,B 0,C 180,E1 6613.924,E2 6613.924} C_VEL
LIN {X 0,Y 473.999,Z 691.44,A -85,B 0,C 180,E1 6623.678,E2 6623.678} C_VEL
LIN {X 0,Y 474.248,Z 691.44,A -85,B 0,C 180,E1 6632.351,E2 6632.351} C_VEL
LIN {X 0,Y 474.983,Z 691.44,A -85,B 0,C 180,E1 6644.235,E2 6644.235} C_VEL
LIN {X 0,Y 475.086,Z 691.44,A -85,B 0,C 180,E1 6653.571,E2 6653.571} C_VEL
LIN {X 0,Y 475.158,Z 691.44,A -85,B 0,C 180,E1 6662.733,E2 6662.733} C_VEL
LIN {X 0,Y 474.66,Z 691.44,A -85,B 0,C 180,E1 6672.798,E2 6672.798} C_VEL
LIN {X 0,Y 474.494,Z 691.44,A -85,B 0,C 180,E1 6681.559,E2 6681.559} C_VEL
LIN {X 0,Y 474.116,Z 691.44,A -85,B 0,C 180,E1 6691.979,E2 6691.979} C_VEL
LIN {X 0,Y 474.014,Z 691.44,A -85,B 0,C 180,E1 6701.203,E2 6701.203} C_VEL
LIN {X 0,Y 474.364,Z 693.407,A -85,B 0,C 180,E1 6704.893,E2 6704.893} C_VEL
LIN {X 0,Y 501.822,Z 745.402,A -85,B 0,C 180,E1 6708.929,E2 6708.929} C_VEL
LIN {X 0,Y 498.929,Z 791.931,A -85,B 0,C 180,E1 6710.391,E2 6710.391} C_VEL
LIN {X 0,Y 489.601,Z 824.975,A -85,B 0,C 180,E1 6711.434,E2 6711.434} C_VEL
LIN {X 0,Y 482.23,Z 885.8,A -85,B 0,C 180,E1 6715.91,E2 6715.91} C_VEL
LIN {X 0,Y 474.752,Z 938.782,A -85,B 0,C 180,E1 6722.106,E2 6722.106} C_VEL
LIN {X 0,Y 469.789,Z 979.334,A -85,B 0,C 180,E1 6729.407,E2 6729.407} C_VEL
LIN {X 0,Y 467.579,Z 1006.517,A -85,B 0,C 180,E1 6737.181,E2 6737.181} C_VEL
LIN {X 0,Y 467.427,Z 1020.766,A -85,B 0,C 180,E1 6745.344,E2 6745.344} C_VEL
LIN {X 0,Y 467.24,Z 1022.149,A -85,B 0,C 180,E1 6752.792,E2 6752.792} C_VEL
LIN {X 0,Y 467.127,Z 1012.357,A -85,B 0,C 180,E1 6760.293,E2 6760.293} C_VEL
LIN {X 0,Y 468.534,Z 991.96,A -85,B 0,C 180,E1 6767.47,E2 6767.47} C_VEL
LIN {X 0,Y 472.357,Z 957.345,A -85,B 0,C 180,E1 6774.94,E2 6774.94} C_VEL
LIN {X 0,Y 478.967,Z 908.495,A -85,B 0,C 180,E1 6781.766,E2 6781.766} C_VEL
LIN {X 0,Y 486.39,Z 852.855,A -85,B 0,C 180,E1 6786.774,E2 6786.774} C_VEL
LIN {X 0,Y 492.882,Z 789.156,A -85,B 0,C 180,E1 6790.285,E2 6790.285} C_VEL
LIN {X 0,Y 494.369,Z 742.296,A -85,B 0,C 180,E1 6791.867,E2 6791.867} C_VEL
LIN {X 0,Y 466.119,Z 691.44,A -85,B 0,C 180,E1 6796.404,E2 6796.404} C_VEL
LIN {X 0,Y 466.049,Z 691.44,A -85,B 0,C 180,E1 6807.529,E2 6807.529} C_VEL
LIN {X 0,Y 466.098,Z 691.44,A -85,B 0,C 180,E1 6816.007,E2 6816.007} C_VEL
LIN {X 0,Y 466.437,Z 691.44,A -85,B 0,C 180,E1 6825.894,E2 6825.894} C_VEL
LIN {X 0,Y 466.833,Z 691.44,A -85,B 0,C 180,E1 6835.353,E2 6835.353} C_VEL
LIN {X 0,Y 466.824,Z 691.44,A -85,B 0,C 180,E1 6842.807,E2 6842.807} C_VEL
LIN {X 0,Y 466.827,Z 691.44,A -85,B 0,C 180,E1 6852.207,E2 6852.207} C_VEL
LIN {X 0,Y 466.75,Z 692.992,A -85,B 0,C 180,E1 6856.467,E2 6856.467} C_VEL
LIN {X 0,Y 494.12,Z 747.735,A -85,B 0,C 180,E1 6861.181,E2 6861.181} C_VEL
LIN {X 0,Y 487.677,Z 813.343,A -85,B 0,C 180,E1 6864.45,E2 6864.45} C_VEL
LIN {X 0,Y 480.103,Z 871.347,A -85,B 0,C 180,E1 6869.421,E2 6869.421} C_VEL
LIN {X 0,Y 473.595,Z 919.736,A -85,B 0,C 180,E1 6875.768,E2 6875.768} C_VEL
LIN {X 0,Y 469.556,Z 957.579,A -85,B 0,C 180,E1 6883.349,E2 6883.349} C_VEL
LIN {X 0,Y 467.393,Z 982.653,A -85,B 0,C 180,E1 6891.788,E2 6891.788} C_VEL
LIN {X 0,Y 466.657,Z 992.35,A -85,B 0,C 180,E1 6899.509,E2 6899.509} C_VEL
LIN {X 0,Y 467.222,Z 989.602,A -85,B 0,C 180,E1 6907.76,E2 6907.76} C_VEL
LIN {X 0,Y 468.233,Z 973.269,A -85,B 0,C 180,E1 6915.932,E2 6915.932} C_VEL
LIN {X 0,Y 470.766,Z 942.617,A -85,B 0,C 180,E1 6923.987,E2 6923.987} C_VEL
LIN {X 0,Y 476.506,Z 897.7,A -85,B 0,C 180,E1 6931.369,E2 6931.369} C_VEL
LIN {X 0,Y 484.208,Z 841.597,A -85,B 0,C 180,E1 6937.315,E2 6937.315} C_VEL
LIN {X 0,Y 491.127,Z 780.568,A -85,B 0,C 180,E1 6941.361,E2 6941.361} C_VEL
LIN {X 0,Y 492.978,Z 742.155,A -85,B 0,C 180,E1 6943.077,E2 6943.077} C_VEL
LIN {X 0,Y 466.69,Z 691.44,A -85,B 0,C 180,E1 6947.553,E2 6947.553} C_VEL
LIN {X 0,Y 466.272,Z 691.44,A -85,B 0,C 180,E1 6958.16,E2 6958.16} C_VEL
LIN {X 0,Y 465.983,Z 691.44,A -85,B 0,C 180,E1 6967.076,E2 6967.076} C_VEL
LIN {X 0,Y 466.021,Z 691.44,A -85,B 0,C 180,E1 6977.115,E2 6977.115} C_VEL
LIN {X 0,Y 466.106,Z 691.44,A -85,B 0,C 180,E1 6987.503,E2 6987.503} C_VEL
LIN {X 0,Y 466.136,Z 691.44,A -85,B 0,C 180,E1 6995.981,E2 6995.981} C_VEL
LIN {X 0,Y 467.097,Z 691.44,A -85,B 0,C 180,E1 7005.889,E2 7005.889} C_VEL
LIN {X 0,Y 467.009,Z 691.44,A -85,B 0,C 180,E1 7015.329,E2 7015.329} C_VEL
LIN {X 0,Y 467.139,Z 691.44,A -85,B 0,C 180,E1 7022.779,E2 7022.779} C_VEL
LIN {X 0,Y 466.694,Z 691.44,A -85,B 0,C 180,E1 7032.185,E2 7032.185} C_VEL
LIN {X 0,Y 466.442,Z 691.44,A -85,B 0,C 180,E1 7041.987,E2 7041.987} C_VEL
LIN {X 0,Y 466.041,Z 691.44,A -85,B 0,C 180,E1 7052.472,E2 7052.472} C_VEL
LIN {X 0,Y 466.027,Z 691.44,A -85,B 0,C 180,E1 7063.594,E2 7063.594} C_VEL
LIN {X 0,Y 495.622,Z 747.104,A -85,B 0,C 180,E1 7068.371,E2 7068.371} C_VEL
LIN {X 0,Y 490.912,Z 812.153,A -85,B 0,C 180,E1 7070.745,E2 7070.745} C_VEL
LIN {X 0,Y 489.601,Z 824.975,A -85,B 0,C 180,E1 7071.434,E2 7071.434} C_VEL
LIN {X 0,Y 479.164,Z 856.48,A -85,B 0,C 180,E1 7072.901,E2 7072.901} C_VEL
LIN {X 0,Y 471.218,Z 914.038,A -85,B 0,C 180,E1 7078.365,E2 7078.365} C_VEL
LIN {X 0,Y 464.815,Z 960.052,A -85,B 0,C 180,E1 7085.142,E2 7085.142} C_VEL
LIN {X 0,Y 460.742,Z 994.921,A -85,B 0,C 180,E1 7093.065,E2 7093.065} C_VEL
LIN {X 0,Y 459.355,Z 1014.285,A -85,B 0,C 180,E1 7100.491,E2 7100.491} C_VEL
LIN {X 0,Y 459.036,Z 1022.148,A -85,B 0,C 180,E1 7107.157,E2 7107.157} C_VEL
LIN {X 0,Y 459.05,Z 1020.767,A -85,B 0,C 180,E1 7114.74,E2 7114.74} C_VEL
LIN {X 0,Y 459.43,Z 1008.073,A -85,B 0,C 180,E1 7122.398,E2 7122.398} C_VEL
LIN {X 0,Y 462.106,Z 980.887,A -85,B 0,C 180,E1 7130.591,E2 7130.591} C_VEL
LIN {X 0,Y 467.679,Z 938.877,A -85,B 0,C 180,E1 7138.339,E2 7138.339} C_VEL
LIN {X 0,Y 475.028,Z 887.067,A -85,B 0,C 180,E1 7144.491,E2 7144.491} C_VEL
LIN {X 0,Y 482.893,Z 825.603,A -85,B 0,C 180,E1 7149.101,E2 7149.101} C_VEL
LIN {X 0,Y 488.959,Z 760.202,A -85,B 0,C 180,E1 7151.858,E2 7151.858} C_VEL
LIN {X 0,Y 487.769,Z 744.628,A -85,B 0,C 180,E1 7152.468,E2 7152.468} C_VEL
LIN {X 0,Y 458.023,Z 691.44,A -85,B 0,C 180,E1 7157.253,E2 7157.253} C_VEL
LIN {X 0,Y 458.048,Z 691.44,A -85,B 0,C 180,E1 7167.656,E2 7167.656} C_VEL
LIN {X 0,Y 457.953,Z 691.44,A -85,B 0,C 180,E1 7177.621,E2 7177.621} C_VEL
LIN {X 0,Y 458.418,Z 691.44,A -85,B 0,C 180,E1 7187.592,E2 7187.592} C_VEL
LIN {X 0,Y 459.12,Z 691.44,A -85,B 0,C 180,E1 7197.172,E2 7197.172} C_VEL
LIN {X 0,Y 459.079,Z 691.44,A -85,B 0,C 180,E1 7206.655,E2 7206.655} C_VEL
LIN {X 0,Y 458.69,Z 692.418,A -85,B 0,C 180,E1 7215.417,E2 7215.417} C_VEL
LIN {X 0,Y 487.78,Z 749.425,A -85,B 0,C 180,E1 7220.612,E2 7220.612} C_VEL
LIN {X 0,Y 481.095,Z 814.564,A -85,B 0,C 180,E1 7223.929,E2 7223.929} C_VEL
LIN {X 0,Y 472.958,Z 872.667,A -85,B 0,C 180,E1 7229.014,E2 7229.014} C_VEL
LIN {X 0,Y 465.859,Z 921.908,A -85,B 0,C 180,E1 7235.673,E2 7235.673} C_VEL
LIN {X 0,Y 461.399,Z 959.921,A -85,B 0,C 180,E1 7243.623,E2 7243.623} C_VEL
LIN {X 0,Y 459.48,Z 982.613,A -85,B 0,C 180,E1 7251.589,E2 7251.589} C_VEL
LIN {X 0,Y 458.666,Z 992.193,A -85,B 0,C 180,E1 7259.147,E2 7259.147} C_VEL
LIN {X 0,Y 458.833,Z 991.725,A -85,B 0,C 180,E1 7265.579,E2 7265.579} C_VEL
LIN {X 0,Y 459.467,Z 979.682,A -85,B 0,C 180,E1 7273.695,E2 7273.695} C_VEL
LIN {X 0,Y 461.928,Z 953.32,A -85,B 0,C 180,E1 7281.974,E2 7281.974} C_VEL
LIN {X 0,Y 467.24,Z 912.282,A -85,B 0,C 180,E1 7289.768,E2 7289.768} C_VEL
LIN {X 0,Y 474.766,Z 860.088,A -85,B 0,C 180,E1 7296.211,E2 7296.211} C_VEL
LIN {X 0,Y 482.842,Z 800.523,A -85,B 0,C 180,E1 7300.87,E2 7300.87} C_VEL
LIN {X 0,Y 486.751,Z 745.56,A -85,B 0,C 180,E1 7303.581,E2 7303.581} C_VEL
LIN {X 0,Y 458.536,Z 691.44,A -85,B 0,C 180,E1 7308.593,E2 7308.593} C_VEL
LIN {X 0,Y 458.222,Z 691.44,A -85,B 0,C 180,E1 7318.701,E2 7318.701} C_VEL
LIN {X 0,Y 457.954,Z 691.44,A -85,B 0,C 180,E1 7328.858,E2 7328.858} C_VEL
LIN {X 0,Y 457.986,Z 691.44,A -85,B 0,C 180,E1 7338.208,E2 7338.208} C_VEL
LIN {X 0,Y 458.071,Z 691.44,A -85,B 0,C 180,E1 7349.099,E2 7349.099} C_VEL
LIN {X 0,Y 457.966,Z 691.44,A -85,B 0,C 180,E1 7357.594,E2 7357.594} C_VEL
LIN {X 0,Y 458.969,Z 691.44,A -85,B 0,C 180,E1 7367.58,E2 7367.58} C_VEL
LIN {X 0,Y 458.838,Z 691.44,A -85,B 0,C 180,E1 7377.144,E2 7377.144} C_VEL
LIN {X 0,Y 458.812,Z 691.44,A -85,B 0,C 180,E1 7384.729,E2 7384.729} C_VEL
LIN {X 0,Y 458.702,Z 691.44,A -85,B 0,C 180,E1 7394.349,E2 7394.349} C_VEL
LIN {X 0,Y 458.324,Z 691.44,A -85,B 0,C 180,E1 7404.426,E2 7404.426} C_VEL
LIN {X 0,Y 457.988,Z 691.44,A -85,B 0,C 180,E1 7413.115,E2 7413.115} C_VEL
LIN {X 0,Y 458.102,Z 692.918,A -85,B 0,C 180,E1 7422.869,E2 7422.869} C_VEL
LIN {X 0,Y 489.39,Z 750.411,A -85,B 0,C 180,E1 7427.839,E2 7427.839} C_VEL
LIN {X 0,Y 484.294,Z 815.014,A -85,B 0,C 180,E1 7430.3,E2 7430.3} C_VEL
LIN {X 0,Y 479.164,Z 856.48,A -85,B 0,C 180,E1 7432.901,E2 7432.901} C_VEL
LIN {X 0,Y 468.305,Z 886.117,A -85,B 0,C 180,E1 7434.87,E2 7434.87} C_VEL
LIN {X 0,Y 460.024,Z 939.191,A -85,B 0,C 180,E1 7441.197,E2 7441.197} C_VEL
LIN {X 0,Y 454.237,Z 979.526,A -85,B 0,C 180,E1 7448.714,E2 7448.714} C_VEL
LIN {X 0,Y 451.618,Z 1006.089,A -85,B 0,C 180,E1 7456.547,E2 7456.547} C_VEL
LIN {X 0,Y 451.243,Z 1019.889,A -85,B 0,C 180,E1 7464.209,E2 7464.209} C_VEL
LIN {X 0,Y 451.213,Z 1022.149,A -85,B 0,C 180,E1 7472.891,E2 7472.891} C_VEL
LIN {X 0,Y 451.149,Z 1012.357,A -85,B 0,C 180,E1 7480.661,E2 7480.661} C_VEL
LIN {X 0,Y 452.829,Z 991.615,A -85,B 0,C 180,E1 7488.196,E2 7488.196} C_VEL
LIN {X 0,Y 457.264,Z 957.341,A -85,B 0,C 180,E1 7495.823,E2 7495.823} C_VEL
LIN {X 0,Y 464.53,Z 909.983,A -85,B 0,C 180,E1 7502.618,E2 7502.618} C_VEL
LIN {X 0,Y 473.155,Z 851.894,A -85,B 0,C 180,E1 7507.97,E2 7507.97} C_VEL
LIN {X 0,Y 480.475,Z 788.933,A -85,B 0,C 180,E1 7511.492,E2 7511.492} C_VEL
LIN {X 0,Y 482.125,Z 748.795,A -85,B 0,C 180,E1 7512.932,E2 7512.932} C_VEL
LIN {X 0,Y 450.006,Z 691.44,A -85,B 0,C 180,E1 7518.512,E2 7518.512} C_VEL
LIN {X 0,Y 450.056,Z 691.44,A -85,B 0,C 180,E1 7529.3,E2 7529.3} C_VEL
LIN {X 0,Y 449.959,Z 691.44,A -85,B 0,C 180,E1 7539.281,E2 7539.281} C_VEL
LIN {X 0,Y 450.62,Z 691.44,A -85,B 0,C 180,E1 7549.343,E2 7549.343} C_VEL
